LIN {X 0,Y 254.905,Z 183.243,A -85,B 0,C 180,E1 -18881.826,E2 -18881.826} C_VEL
LIN {X 0,Y 256.639,Z 184.875,A -85,B 0,C 180,E1 -18883.002,E2 -18883.002} C_VEL
LIN {X 0,Y 260.021,Z 189.343,A -85,B 0,C 180,E1 -18885.127,E2 -18885.127} C_VEL
LIN {X 0,Y 261.601,Z 191.447,A -85,B 0,C 180,E1 -18886.008,E2 -18886.008} C_VEL
LIN {X 0,Y 265.009,Z 196.05,A -85,B 0,C 180,E1 -18887.751,E2 -18887.751} C_VEL
LIN {X 0,Y 268.493,Z 201.125,A -85,B 0,C 180,E1 -18889.357,E2 -18889.357} C_VEL
LIN {X 0,Y 271.454,Z 205.94,A -85,B 0,C 180,E1 -18890.618,E2 -18890.618} C_VEL
LIN {X 0,Y 277.657,Z 217.044,A -85,B 0,C 180,E1 -18893.04,E2 -18893.04} C_VEL
LIN {X 0,Y 281.725,Z 226.048,A -85,B 0,C 180,E1 -18894.546,E2 -18894.546} C_VEL
LIN {X 0,Y 276.676,Z 285.05,A -85,B 0,C 180,E1 -18896.614,E2 -18896.614} C_VEL
LIN {X 0,Y 274.99,Z 297.648,A -85,B 0,C 180,E1 -18897.29,E2 -18897.29} C_VEL
LIN {X 0,Y 273.026,Z 309.594,A -85,B 0,C 180,E1 -18898.211,E2 -18898.211} C_VEL
LIN {X 0,Y 270.772,Z 320.185,A -85,B 0,C 180,E1 -18899.257,E2 -18899.257} C_VEL
LIN {X 0,Y 267.635,Z 332.608,A -85,B 0,C 180,E1 -18900.856,E2 -18900.856} C_VEL
LIN {X 0,Y 264.368,Z 343.674,A -85,B 0,C 180,E1 -18902.667,E2 -18902.667} C_VEL
LIN {X 0,Y 260.959,Z 353.865,A -85,B 0,C 180,E1 -18904.808,E2 -18904.808} C_VEL
LIN {X 0,Y 258.393,Z 360.832,A -85,B 0,C 180,E1 -18906.638,E2 -18906.638} C_VEL
LIN {X 0,Y 255.598,Z 368.03,A -85,B 0,C 180,E1 -18908.991,E2 -18908.991} C_VEL
LIN {X 0,Y 253.363,Z 373.364,A -85,B 0,C 180,E1 -18911.197,E2 -18911.197} C_VEL
LIN {X 0,Y 251.204,Z 378.159,A -85,B 0,C 180,E1 -18913.758,E2 -18913.758} C_VEL
LIN {X 0,Y 249.407,Z 381.995,A -85,B 0,C 180,E1 -18916.645,E2 -18916.645} C_VEL
LIN {X 0,Y 248.021,Z 384.63,A -85,B 0,C 180,E1 -18919.88,E2 -18919.88} C_VEL
LIN {X 0,Y 247.437,Z 385.342,A -85,B 0,C 180,E1 -18921.669,E2 -18921.669} C_VEL
LIN {X 0,Y 246.862,Z 385.521,A -85,B 0,C 180,E1 -18924.351,E2 -18924.351} C_VEL
LIN {X 0,Y 246.591,Z 384.531,A -85,B 0,C 180,E1 -18927.131,E2 -18927.131} C_VEL
LIN {X 0,Y 246.526,Z 383.207,A -85,B 0,C 180,E1 -18928.989,E2 -18928.989} C_VEL
LIN {X 0,Y 246.787,Z 379.889,A -85,B 0,C 180,E1 -18931.942,E2 -18931.942} C_VEL
LIN {X 0,Y 247.195,Z 375.495,A -85,B 0,C 180,E1 -18934.655,E2 -18934.655} C_VEL
LIN {X 0,Y 247.774,Z 369.505,A -85,B 0,C 180,E1 -18937.418,E2 -18937.418} C_VEL
LIN {X 0,Y 248.552,Z 362.739,A -85,B 0,C 180,E1 -18939.841,E2 -18939.841} C_VEL
LIN {X 0,Y 249.449,Z 355.299,A -85,B 0,C 180,E1 -18942.001,E2 -18942.001} C_VEL
LIN {X 0,Y 250.528,Z 346.497,A -85,B 0,C 180,E1 -18944.092,E2 -18944.092} C_VEL
LIN {X 0,Y 251.803,Z 336.515,A -85,B 0,C 180,E1 -18946.013,E2 -18946.013} C_VEL
LIN {X 0,Y 253.278,Z 324.244,A -85,B 0,C 180,E1 -18947.882,E2 -18947.882} C_VEL
LIN {X 0,Y 254.569,Z 312.848,A -85,B 0,C 180,E1 -18949.243,E2 -18949.243} C_VEL
LIN {X 0,Y 255.708,Z 299.284,A -85,B 0,C 180,E1 -18950.473,E2 -18950.473} C_VEL
LIN {X 0,Y 256.538,Z 286.069,A -85,B 0,C 180,E1 -18951.331,E2 -18951.331} C_VEL
LIN {X 0,Y 257.364,Z 267.967,A -85,B 0,C 180,E1 -18952.047,E2 -18952.047} C_VEL
LIN {X 0,Y 259.677,Z 209.083,A -85,B 0,C 180,E1 -18954.102,E2 -18954.102} C_VEL
LIN {X 0,Y 258.379,Z 202.077,A -85,B 0,C 180,E1 -18954.456,E2 -18954.456} C_VEL
LIN {X 0,Y 249.422,Z 174.029,A -85,B 0,C 180,E1 -18956.245,E2 -18956.245} C_VEL
LIN {X 0,Y 249.088,Z 172.457,A -85,B 0,C 180,E1 -18956.92,E2 -18956.92} C_VEL
LIN {X 0,Y 249.039,Z 172.462,A -85,B 0,C 180,E1 -18961.33,E2 -18961.33} C_VEL
LIN {X 0,Y 249.06,Z 172.46,A -85,B 0,C 180,E1 -18964.957,E2 -18964.957} C_VEL
LIN {X 0,Y 249.055,Z 172.461,A -85,B 0,C 180,E1 -18968.627,E2 -18968.627} C_VEL
LIN {X 0,Y 249.162,Z 172.448,A -85,B 0,C 180,E1 -18973.615,E2 -18973.615} C_VEL
LIN {X 0,Y 249.223,Z 172.44,A -85,B 0,C 180,E1 -18978.614,E2 -18978.614} C_VEL
LIN {X 0,Y 249.435,Z 172.416,A -85,B 0,C 180,E1 -18981.9,E2 -18981.9} C_VEL
LIN {X 0,Y 249.264,Z 172.434,A -85,B 0,C 180,E1 -18985.146,E2 -18985.146} C_VEL
LIN {X 0,Y 249.661,Z 172.384,A -85,B 0,C 180,E1 -18988.386,E2 -18988.386} C_VEL
LIN {X 0,Y 249.66,Z 172.385,A -85,B 0,C 180,E1 -18991.612,E2 -18991.612} C_VEL
LIN {X 0,Y 249.428,Z 172.412,A -85,B 0,C 180,E1 -18996.47,E2 -18996.47} C_VEL
LIN {X 0,Y 249.335,Z 172.427,A -85,B 0,C 180,E1 -18999.735,E2 -18999.735} C_VEL
LIN {X 0,Y 249.147,Z 172.448,A -85,B 0,C 180,E1 -19004.705,E2 -19004.705} C_VEL
LIN {X 0,Y 249.079,Z 172.456,A -85,B 0,C 180,E1 -19008.08,E2 -19008.08} C_VEL
LIN {X 0,Y 249.043,Z 172.464,A -85,B 0,C 180,E1 -19011.521,E2 -19011.521} C_VEL
LIN {X 0,Y 249.047,Z 172.462,A -85,B 0,C 180,E1 -19015.44,E2 -19015.44} C_VEL
LIN {X 0,Y 249.036,Z 172.464,A -85,B 0,C 180,E1 -19018.972,E2 -19018.972} C_VEL
LIN {X 0,Y 249.026,Z 172.462,A -85,B 0,C 180,E1 -19022.425,E2 -19022.425} C_VEL
LIN {X 0,Y 249.025,Z 172.463,A -85,B 0,C 180,E1 -19026.344,E2 -19026.344} C_VEL
LIN {X 0,Y 248.976,Z 172.47,A -85,B 0,C 180,E1 -19030.482,E2 -19030.482} C_VEL
LIN {X 0,Y 248.959,Z 172.475,A -85,B 0,C 180,E1 -19034.887,E2 -19034.887} C_VEL
LIN {X 0,Y 248.976,Z 172.47,A -85,B 0,C 180,E1 -19037.353,E2 -19037.353} C_VEL
LIN {X 0,Y 249.036,Z 172.462,A -85,B 0,C 180,E1 -19042.2,E2 -19042.2} C_VEL
LIN {X 0,Y 249.039,Z 172.461,A -85,B 0,C 180,E1 -19045.638,E2 -19045.638} C_VEL
LIN {X 0,Y 248.997,Z 172.465,A -85,B 0,C 180,E1 -19049.465,E2 -19049.465} C_VEL
LIN {X 0,Y 249.016,Z 172.465,A -85,B 0,C 180,E1 -19053.155,E2 -19053.155} C_VEL
LIN {X 0,Y 249,Z 172.466,A -85,B 0,C 180,E1 -19056.724,E2 -19056.724} C_VEL
LIN {X 0,Y 249.037,Z 172.464,A -85,B 0,C 180,E1 -19060.205,E2 -19060.205} C_VEL
LIN {X 0,Y 249.152,Z 172.447,A -85,B 0,C 180,E1 -19063.615,E2 -19063.615} C_VEL
LIN {X 0,Y 249.211,Z 172.441,A -85,B 0,C 180,E1 -19068.614,E2 -19068.614} C_VEL
LIN {X 0,Y 249.425,Z 172.416,A -85,B 0,C 180,E1 -19071.901,E2 -19071.901} C_VEL
LIN {X 0,Y 249.254,Z 172.433,A -85,B 0,C 180,E1 -19075.147,E2 -19075.147} C_VEL
LIN {X 0,Y 249.65,Z 172.387,A -85,B 0,C 180,E1 -19078.386,E2 -19078.386} C_VEL
LIN {X 0,Y 249.649,Z 172.386,A -85,B 0,C 180,E1 -19081.613,E2 -19081.613} C_VEL
LIN {X 0,Y 249.418,Z 172.415,A -85,B 0,C 180,E1 -19086.471,E2 -19086.471} C_VEL
LIN {X 0,Y 249.325,Z 172.428,A -85,B 0,C 180,E1 -19089.737,E2 -19089.737} C_VEL
LIN {X 0,Y 249.138,Z 172.449,A -85,B 0,C 180,E1 -19094.707,E2 -19094.707} C_VEL
LIN {X 0,Y 249.119,Z 172.448,A -85,B 0,C 180,E1 -19095.622,E2 -19095.622} C_VEL
LIN {X 0,Y 248.461,Z 172.535,A -85,B 0,C 180,E1 -19096.971,E2 -19096.971} C_VEL
LIN {X 0,Y 245.577,Z 172.894,A -85,B 0,C 180,E1 -19099.169,E2 -19099.169} C_VEL
LIN {X 0,Y 243.104,Z 173.201,A -85,B 0,C 180,E1 -19100.959,E2 -19100.959} C_VEL
LIN {X 0,Y 242.028,Z 173.335,A -85,B 0,C 180,E1 -19102.349,E2 -19102.349} C_VEL
LIN {X 0,Y 241.933,Z 173.344,A -85,B 0,C 180,E1 -19102.821,E2 -19102.821} C_VEL
LIN {X 0,Y 241.98,Z 173.341,A -85,B 0,C 180,E1 -19105.827,E2 -19105.827} C_VEL
LIN {X 0,Y 241.962,Z 173.345,A -85,B 0,C 180,E1 -19109.589,E2 -19109.589} C_VEL
LIN {X 0,Y 241.973,Z 173.343,A -85,B 0,C 180,E1 -19113.494,E2 -19113.494} C_VEL
LIN {X 0,Y 241.977,Z 173.342,A -85,B 0,C 180,E1 -19117.584,E2 -19117.584} C_VEL
LIN {X 0,Y 241.902,Z 173.35,A -85,B 0,C 180,E1 -19121.93,E2 -19121.93} C_VEL
LIN {X 0,Y 241.895,Z 173.354,A -85,B 0,C 180,E1 -19126.581,E2 -19126.581} C_VEL
LIN {X 0,Y 241.988,Z 173.34,A -85,B 0,C 180,E1 -19131.642,E2 -19131.642} C_VEL
LIN {X 0,Y 242.069,Z 173.515,A -85,B 0,C 180,E1 -19136.148,E2 -19136.148} C_VEL
LIN {X 0,Y 244.15,Z 184.245,A -85,B 0,C 180,E1 -19140.267,E2 -19140.267} C_VEL
LIN {X 0,Y 244.801,Z 187.444,A -85,B 0,C 180,E1 -19141.446,E2 -19141.446} C_VEL
LIN {X 0,Y 248.272,Z 199.557,A -85,B 0,C 180,E1 -19142.193,E2 -19142.193} C_VEL
LIN {X 0,Y 252.252,Z 234.822,A -85,B 0,C 180,E1 -19143.86,E2 -19143.86} C_VEL
LIN {X 0,Y 249.825,Z 295.765,A -85,B 0,C 180,E1 -19146.093,E2 -19146.093} C_VEL
LIN {X 0,Y 248.844,Z 309.841,A -85,B 0,C 180,E1 -19146.931,E2 -19146.931} C_VEL
LIN {X 0,Y 247.722,Z 321.604,A -85,B 0,C 180,E1 -19147.921,E2 -19147.921} C_VEL
LIN {X 0,Y 246.377,Z 334.101,A -85,B 0,C 180,E1 -19149.331,E2 -19149.331} C_VEL
LIN {X 0,Y 244.925,Z 345.362,A -85,B 0,C 180,E1 -19150.951,E2 -19150.951} C_VEL
LIN {X 0,Y 243.54,Z 355.921,A -85,B 0,C 180,E1 -19152.864,E2 -19152.864} C_VEL
LIN {X 0,Y 242.419,Z 364.893,A -85,B 0,C 180,E1 -19154.877,E2 -19154.877} C_VEL
LIN {X 0,Y 241.251,Z 373.932,A -85,B 0,C 180,E1 -19157.381,E2 -19157.381} C_VEL
LIN {X 0,Y 240.534,Z 381.125,A -85,B 0,C 180,E1 -19159.905,E2 -19159.905} C_VEL
LIN {X 0,Y 240.116,Z 386.836,A -85,B 0,C 180,E1 -19162.433,E2 -19162.433} C_VEL
LIN {X 0,Y 239.919,Z 391.263,A -85,B 0,C 180,E1 -19164.96,E2 -19164.96} C_VEL
LIN {X 0,Y 239.892,Z 393.581,A -85,B 0,C 180,E1 -19166.642,E2 -19166.642} C_VEL
LIN {X 0,Y 239.92,Z 395.406,A -85,B 0,C 180,E1 -19168.323,E2 -19168.323} C_VEL
LIN {X 0,Y 239.916,Z 396.747,A -85,B 0,C 180,E1 -19170.001,E2 -19170.001} C_VEL
LIN {X 0,Y 239.893,Z 397.668,A -85,B 0,C 180,E1 -19171.68,E2 -19171.68} C_VEL
LIN {X 0,Y 239.775,Z 398.264,A -85,B 0,C 180,E1 -19174.748,E2 -19174.748} C_VEL
LIN {X 0,Y 239.96,Z 397.891,A -85,B 0,C 180,E1 -19176.729,E2 -19176.729} C_VEL
LIN {X 0,Y 240.757,Z 396.027,A -85,B 0,C 180,E1 -19180.089,E2 -19180.089} C_VEL
LIN {X 0,Y 241.785,Z 393.519,A -85,B 0,C 180,E1 -19182.593,E2 -19182.593} C_VEL
LIN {X 0,Y 243.188,Z 390.027,A -85,B 0,C 180,E1 -19185.077,E2 -19185.077} C_VEL
LIN {X 0,Y 245.352,Z 385.49,A -85,B 0,C 180,E1 -19187.505,E2 -19187.505} C_VEL
LIN {X 0,Y 248.14,Z 378.736,A -85,B 0,C 180,E1 -19190.302,E2 -19190.302} C_VEL
LIN {X 0,Y 250.933,Z 371.563,A -85,B 0,C 180,E1 -19192.608,E2 -19192.608} C_VEL
LIN {X 0,Y 254.355,Z 362.426,A -85,B 0,C 180,E1 -19194.922,E2 -19194.922} C_VEL
LIN {X 0,Y 257.945,Z 352.315,A -85,B 0,C 180,E1 -19196.936,E2 -19196.936} C_VEL
LIN {X 0,Y 261.529,Z 340.93,A -85,B 0,C 180,E1 -19198.71,E2 -19198.71} C_VEL
LIN {X 0,Y 264.574,Z 329.639,A -85,B 0,C 180,E1 -19200.093,E2 -19200.093} C_VEL
LIN {X 0,Y 267.49,Z 316.966,A -85,B 0,C 180,E1 -19201.26,E2 -19201.26} C_VEL
LIN {X 0,Y 270.042,Z 303.682,A -85,B 0,C 180,E1 -19202.135,E2 -19202.135} C_VEL
LIN {X 0,Y 271.757,Z 289.867,A -85,B 0,C 180,E1 -19202.785,E2 -19202.785} C_VEL
LIN {X 0,Y 275.895,Z 241.621,A -85,B 0,C 180,E1 -19204.522,E2 -19204.522} C_VEL
LIN {X 0,Y 275,Z 233.168,A -85,B 0,C 180,E1 -19205.232,E2 -19205.232} C_VEL
LIN {X 0,Y 271.422,Z 224.233,A -85,B 0,C 180,E1 -19206.741,E2 -19206.741} C_VEL
LIN {X 0,Y 266.748,Z 214.805,A -85,B 0,C 180,E1 -19208.789,E2 -19208.789} C_VEL
LIN {X 0,Y 264.621,Z 210.789,A -85,B 0,C 180,E1 -19209.822,E2 -19209.822} C_VEL
LIN {X 0,Y 262.005,Z 206.304,A -85,B 0,C 180,E1 -19211.117,E2 -19211.117} C_VEL
LIN {X 0,Y 258.799,Z 200.968,A -85,B 0,C 180,E1 -19212.915,E2 -19212.915} C_VEL
LIN {X 0,Y 254.883,Z 194.985,A -85,B 0,C 180,E1 -19215.414,E2 -19215.414} C_VEL
LIN {X 0,Y 250.245,Z 188.473,A -85,B 0,C 180,E1 -19219.227,E2 -19219.227} C_VEL
LIN {X 0,Y 246.767,Z 184.055,A -85,B 0,C 180,E1 -19223.65,E2 -19223.65} C_VEL
LIN {X 0,Y 245.502,Z 182.109,A -85,B 0,C 180,E1 -19227.05,E2 -19227.05} C_VEL
LIN {X 0,Y 245.288,Z 181.573,A -85,B 0,C 180,E1 -19229.269,E2 -19229.269} C_VEL
LIN {X 0,Y 245.694,Z 181.933,A -85,B 0,C 180,E1 -19232.047,E2 -19232.047} C_VEL
LIN {X 0,Y 247.908,Z 184.21,A -85,B 0,C 180,E1 -19236.395,E2 -19236.395} C_VEL
LIN {X 0,Y 250.046,Z 185.965,A -85,B 0,C 180,E1 -19238.785,E2 -19238.785} C_VEL
LIN {X 0,Y 253.178,Z 190.055,A -85,B 0,C 180,E1 -19241.593,E2 -19241.593} C_VEL
LIN {X 0,Y 254.488,Z 191.344,A -85,B 0,C 180,E1 -19242.517,E2 -19242.517} C_VEL
LIN {X 0,Y 258.027,Z 196.028,A -85,B 0,C 180,E1 -19244.837,E2 -19244.837} C_VEL
LIN {X 0,Y 262.472,Z 202.382,A -85,B 0,C 180,E1 -19247.297,E2 -19247.297} C_VEL
LIN {X 0,Y 265.653,Z 207.183,A -85,B 0,C 180,E1 -19248.822,E2 -19248.822} C_VEL
LIN {X 0,Y 268.38,Z 211.88,A -85,B 0,C 180,E1 -19250.079,E2 -19250.079} C_VEL
LIN {X 0,Y 274.089,Z 222.548,A -85,B 0,C 180,E1 -19252.449,E2 -19252.449} C_VEL
LIN {X 0,Y 276.862,Z 228.786,A -85,B 0,C 180,E1 -19253.522,E2 -19253.522} C_VEL
LIN {X 0,Y 271.748,Z 285.239,A -85,B 0,C 180,E1 -19255.55,E2 -19255.55} C_VEL
LIN {X 0,Y 269.887,Z 298.289,A -85,B 0,C 180,E1 -19256.268,E2 -19256.268} C_VEL
LIN {X 0,Y 267.768,Z 310.372,A -85,B 0,C 180,E1 -19257.216,E2 -19257.216} C_VEL
LIN {X 0,Y 265.372,Z 320.961,A -85,B 0,C 180,E1 -19258.284,E2 -19258.284} C_VEL
LIN {X 0,Y 262.265,Z 332.663,A -85,B 0,C 180,E1 -19259.808,E2 -19259.808} C_VEL
LIN {X 0,Y 258.966,Z 343.263,A -85,B 0,C 180,E1 -19261.555,E2 -19261.555} C_VEL
LIN {X 0,Y 255.612,Z 352.681,A -85,B 0,C 180,E1 -19263.53,E2 -19263.53} C_VEL
LIN {X 0,Y 251.986,Z 362.014,A -85,B 0,C 180,E1 -19266.004,E2 -19266.004} C_VEL
LIN {X 0,Y 248.799,Z 369.538,A -85,B 0,C 180,E1 -19268.625,E2 -19268.625} C_VEL
LIN {X 0,Y 245.854,Z 375.898,A -85,B 0,C 180,E1 -19271.543,E2 -19271.543} C_VEL
LIN {X 0,Y 243.79,Z 380.082,A -85,B 0,C 180,E1 -19274.185,E2 -19274.185} C_VEL
LIN {X 0,Y 242.176,Z 383.099,A -85,B 0,C 180,E1 -19276.871,E2 -19276.871} C_VEL
LIN {X 0,Y 241.372,Z 384.47,A -85,B 0,C 180,E1 -19278.681,E2 -19278.681} C_VEL
LIN {X 0,Y 240.58,Z 385.479,A -85,B 0,C 180,E1 -19280.799,E2 -19280.799} C_VEL
LIN {X 0,Y 240.168,Z 385.781,A -85,B 0,C 180,E1 -19282.36,E2 -19282.36} C_VEL
LIN {X 0,Y 239.708,Z 385.624,A -85,B 0,C 180,E1 -19284.645,E2 -19284.645} C_VEL
LIN {X 0,Y 239.532,Z 385.104,A -85,B 0,C 180,E1 -19286.111,E2 -19286.111} C_VEL
LIN {X 0,Y 239.438,Z 383.75,A -85,B 0,C 180,E1 -19288.287,E2 -19288.287} C_VEL
LIN {X 0,Y 239.541,Z 381.245,A -85,B 0,C 180,E1 -19290.839,E2 -19290.839} C_VEL
LIN {X 0,Y 239.971,Z 376.997,A -85,B 0,C 180,E1 -19293.811,E2 -19293.811} C_VEL
LIN {X 0,Y 240.509,Z 371.044,A -85,B 0,C 180,E1 -19296.802,E2 -19296.802} C_VEL
LIN {X 0,Y 241.244,Z 364.525,A -85,B 0,C 180,E1 -19299.339,E2 -19299.339} C_VEL
LIN {X 0,Y 242.257,Z 356.378,A -85,B 0,C 180,E1 -19301.855,E2 -19301.855} C_VEL
LIN {X 0,Y 243.418,Z 347.106,A -85,B 0,C 180,E1 -19304.151,E2 -19304.151} C_VEL
LIN {X 0,Y 244.749,Z 336.839,A -85,B 0,C 180,E1 -19306.201,E2 -19306.201} C_VEL
LIN {X 0,Y 246.095,Z 325.865,A -85,B 0,C 180,E1 -19307.947,E2 -19307.947} C_VEL
LIN {X 0,Y 247.486,Z 313.985,A -85,B 0,C 180,E1 -19309.447,E2 -19309.447} C_VEL
LIN {X 0,Y 248.646,Z 301.024,A -85,B 0,C 180,E1 -19310.693,E2 -19310.693} C_VEL
LIN {X 0,Y 249.585,Z 287.032,A -85,B 0,C 180,E1 -19311.663,E2 -19311.663} C_VEL
LIN {X 0,Y 250.44,Z 270.442,A -85,B 0,C 180,E1 -19312.364,E2 -19312.364} C_VEL
LIN {X 0,Y 252.892,Z 210.015,A -85,B 0,C 180,E1 -19314.539,E2 -19314.539} C_VEL
LIN {X 0,Y 251.787,Z 204.045,A -85,B 0,C 180,E1 -19314.85,E2 -19314.85} C_VEL
LIN {X 0,Y 242.629,Z 175.689,A -85,B 0,C 180,E1 -19316.676,E2 -19316.676} C_VEL
LIN {X 0,Y 242.213,Z 174.177,A -85,B 0,C 180,E1 -19316.819,E2 -19316.819} C_VEL
LIN {X 0,Y 242.034,Z 173.334,A -85,B 0,C 180,E1 -19317.294,E2 -19317.294} C_VEL
LIN {X 0,Y 241.976,Z 173.345,A -85,B 0,C 180,E1 -19320.615,E2 -19320.615} C_VEL
LIN {X 0,Y 242.001,Z 173.342,A -85,B 0,C 180,E1 -19324.196,E2 -19324.196} C_VEL
LIN {X 0,Y 241.99,Z 173.343,A -85,B 0,C 180,E1 -19328.337,E2 -19328.337} C_VEL
LIN {X 0,Y 242.11,Z 173.325,A -85,B 0,C 180,E1 -19333.323,E2 -19333.323} C_VEL
LIN {X 0,Y 242.157,Z 173.322,A -85,B 0,C 180,E1 -19338.277,E2 -19338.277} C_VEL
LIN {X 0,Y 242.385,Z 173.292,A -85,B 0,C 180,E1 -19341.663,E2 -19341.663} C_VEL
LIN {X 0,Y 242.404,Z 173.289,A -85,B 0,C 180,E1 -19343.339,E2 -19343.339} C_VEL
LIN {X 0,Y 242.621,Z 173.261,A -85,B 0,C 180,E1 -19348.339,E2 -19348.339} C_VEL
LIN {X 0,Y 242.62,Z 173.263,A -85,B 0,C 180,E1 -19351.658,E2 -19351.658} C_VEL
LIN {X 0,Y 242.398,Z 173.288,A -85,B 0,C 180,E1 -19356.658,E2 -19356.658} C_VEL
LIN {X 0,Y 242.262,Z 173.306,A -85,B 0,C 180,E1 -19360.022,E2 -19360.022} C_VEL
LIN {X 0,Y 242.106,Z 173.326,A -85,B 0,C 180,E1 -19365.143,E2 -19365.143} C_VEL
LIN {X 0,Y 242.017,Z 173.335,A -85,B 0,C 180,E1 -19368.627,E2 -19368.627} C_VEL
LIN {X 0,Y 241.973,Z 173.341,A -85,B 0,C 180,E1 -19372.182,E2 -19372.182} C_VEL
LIN {X 0,Y 241.987,Z 173.339,A -85,B 0,C 180,E1 -19375.825,E2 -19375.825} C_VEL
LIN {X 0,Y 241.968,Z 173.344,A -85,B 0,C 180,E1 -19379.587,E2 -19379.587} C_VEL
LIN {X 0,Y 241.978,Z 173.341,A -85,B 0,C 180,E1 -19383.491,E2 -19383.491} C_VEL
LIN {X 0,Y 241.981,Z 173.342,A -85,B 0,C 180,E1 -19387.581,E2 -19387.581} C_VEL
LIN {X 0,Y 241.905,Z 173.347,A -85,B 0,C 180,E1 -19391.927,E2 -19391.927} C_VEL
LIN {X 0,Y 241.897,Z 173.354,A -85,B 0,C 180,E1 -19396.578,E2 -19396.578} C_VEL
LIN {X 0,Y 241.988,Z 173.339,A -85,B 0,C 180,E1 -19401.64,E2 -19401.64} C_VEL
LIN {X 0,Y 241.975,Z 173.344,A -85,B 0,C 180,E1 -19404.486,E2 -19404.486} C_VEL
LIN {X 0,Y 241.948,Z 173.346,A -85,B 0,C 180,E1 -19408.475,E2 -19408.475} C_VEL
LIN {X 0,Y 241.955,Z 173.346,A -85,B 0,C 180,E1 -19412.306,E2 -19412.306} C_VEL
LIN {X 0,Y 241.976,Z 173.342,A -85,B 0,C 180,E1 -19416.007,E2 -19416.007} C_VEL
LIN {X 0,Y 241.977,Z 173.341,A -85,B 0,C 180,E1 -19419.602,E2 -19419.602} C_VEL
LIN {X 0,Y 242.1,Z 173.325,A -85,B 0,C 180,E1 -19423.323,E2 -19423.323} C_VEL
LIN {X 0,Y 242.145,Z 173.324,A -85,B 0,C 180,E1 -19428.277,E2 -19428.277} C_VEL
LIN {X 0,Y 242.374,Z 173.293,A -85,B 0,C 180,E1 -19431.663,E2 -19431.663} C_VEL
LIN {X 0,Y 242.393,Z 173.288,A -85,B 0,C 180,E1 -19433.34,E2 -19433.34} C_VEL
LIN {X 0,Y 242.61,Z 173.264,A -85,B 0,C 180,E1 -19438.34,E2 -19438.34} C_VEL
LIN {X 0,Y 242.609,Z 173.264,A -85,B 0,C 180,E1 -19441.66,E2 -19441.66} C_VEL
LIN {X 0,Y 242.389,Z 173.29,A -85,B 0,C 180,E1 -19446.66,E2 -19446.66} C_VEL
LIN {X 0,Y 242.253,Z 173.306,A -85,B 0,C 180,E1 -19450.024,E2 -19450.024} C_VEL
LIN {X 0,Y 242.097,Z 173.327,A -85,B 0,C 180,E1 -19455.145,E2 -19455.145} C_VEL
LIN {X 0,Y 242.009,Z 173.335,A -85,B 0,C 180,E1 -19458.629,E2 -19458.629} C_VEL
LIN {X 0,Y 241.933,Z 173.344,A -85,B 0,C 180,E1 -19462.821,E2 -19462.821} C_VEL
LIN {X 0,Y 241.254,Z 173.432,A -85,B 0,C 180,E1 -19464.209,E2 -19464.209} C_VEL
LIN {X 0,Y 238.431,Z 173.781,A -85,B 0,C 180,E1 -19466.475,E2 -19466.475} C_VEL
LIN {X 0,Y 236.033,Z 174.082,A -85,B 0,C 180,E1 -19468.321,E2 -19468.321} C_VEL
LIN {X 0,Y 234.991,Z 174.213,A -85,B 0,C 180,E1 -19469.752,E2 -19469.752} C_VEL
LIN {X 0,Y 234.898,Z 174.223,A -85,B 0,C 180,E1 -19470.237,E2 -19470.237} C_VEL
LIN {X 0,Y 234.935,Z 174.222,A -85,B 0,C 180,E1 -19473.114,E2 -19473.114} C_VEL
LIN {X 0,Y 234.909,Z 174.219,A -85,B 0,C 180,E1 -19476.752,E2 -19476.752} C_VEL
LIN {X 0,Y 234.906,Z 174.224,A -85,B 0,C 180,E1 -19478.936,E2 -19478.936} C_VEL
LIN {X 0,Y 234.848,Z 174.231,A -85,B 0,C 180,E1 -19483.495,E2 -19483.495} C_VEL
LIN {X 0,Y 234.848,Z 174.231,A -85,B 0,C 180,E1 -19486.507,E2 -19486.507} C_VEL
LIN {X 0,Y 234.913,Z 174.224,A -85,B 0,C 180,E1 -19491.08,E2 -19491.08} C_VEL
LIN {X 0,Y 234.974,Z 174.215,A -85,B 0,C 180,E1 -19495.742,E2 -19495.742} C_VEL
LIN {X 0,Y 236.966,Z 184.264,A -85,B 0,C 180,E1 -19499.724,E2 -19499.724} C_VEL
LIN {X 0,Y 237.523,Z 187.283,A -85,B 0,C 180,E1 -19500.863,E2 -19500.863} C_VEL
LIN {X 0,Y 241.639,Z 201.481,A -85,B 0,C 180,E1 -19501.776,E2 -19501.776} C_VEL
LIN {X 0,Y 245.429,Z 235.077,A -85,B 0,C 180,E1 -19503.419,E2 -19503.419} C_VEL
LIN {X 0,Y 242.873,Z 296.425,A -85,B 0,C 180,E1 -19505.763,E2 -19505.763} C_VEL
LIN {X 0,Y 241.803,Z 310.913,A -85,B 0,C 180,E1 -19506.673,E2 -19506.673} C_VEL
LIN {X 0,Y 240.408,Z 324.215,A -85,B 0,C 180,E1 -19507.892,E2 -19507.892} C_VEL
LIN {X 0,Y 239.075,Z 336.161,A -85,B 0,C 180,E1 -19509.345,E2 -19509.345} C_VEL
LIN {X 0,Y 237.67,Z 346.965,A -85,B 0,C 180,E1 -19511.019,E2 -19511.019} C_VEL
LIN {X 0,Y 236.276,Z 357.877,A -85,B 0,C 180,E1 -19513.143,E2 -19513.143} C_VEL
LIN {X 0,Y 235.101,Z 366.753,A -85,B 0,C 180,E1 -19515.282,E2 -19515.282} C_VEL
LIN {X 0,Y 233.99,Z 375.327,A -85,B 0,C 180,E1 -19517.865,E2 -19517.865} C_VEL
LIN {X 0,Y 233.339,Z 382.22,A -85,B 0,C 180,E1 -19520.466,E2 -19520.466} C_VEL
LIN {X 0,Y 232.974,Z 387.672,A -85,B 0,C 180,E1 -19523.071,E2 -19523.071} C_VEL
LIN {X 0,Y 232.779,Z 392.073,A -85,B 0,C 180,E1 -19525.832,E2 -19525.832} C_VEL
LIN {X 0,Y 232.853,Z 394.895,A -85,B 0,C 180,E1 -19528.272,E2 -19528.272} C_VEL
LIN {X 0,Y 232.849,Z 396.323,A -85,B 0,C 180,E1 -19530.001,E2 -19530.001} C_VEL
LIN {X 0,Y 232.822,Z 397.301,A -85,B 0,C 180,E1 -19531.731,E2 -19531.731} C_VEL
LIN {X 0,Y 232.731,Z 398.041,A -85,B 0,C 180,E1 -19535.199,E2 -19535.199} C_VEL
LIN {X 0,Y 232.898,Z 397.786,A -85,B 0,C 180,E1 -19536.934,E2 -19536.934} C_VEL
LIN {X 0,Y 233.754,Z 396.054,A -85,B 0,C 180,E1 -19540.394,E2 -19540.394} C_VEL
LIN {X 0,Y 234.424,Z 394.601,A -85,B 0,C 180,E1 -19542.116,E2 -19542.116} C_VEL
LIN {X 0,Y 235.807,Z 391.606,A -85,B 0,C 180,E1 -19544.676,E2 -19544.676} C_VEL
LIN {X 0,Y 237.807,Z 387.594,A -85,B 0,C 180,E1 -19547.191,E2 -19547.191} C_VEL
LIN {X 0,Y 240.226,Z 382.472,A -85,B 0,C 180,E1 -19549.662,E2 -19549.662} C_VEL
LIN {X 0,Y 243.347,Z 375.051,A -85,B 0,C 180,E1 -19552.455,E2 -19552.455} C_VEL
LIN {X 0,Y 246.815,Z 366.854,A -85,B 0,C 180,E1 -19554.836,E2 -19554.836} C_VEL
LIN {X 0,Y 250.079,Z 358.685,A -85,B 0,C 180,E1 -19556.723,E2 -19556.723} C_VEL
LIN {X 0,Y 253.618,Z 348.854,A -85,B 0,C 180,E1 -19558.557,E2 -19558.557} C_VEL
LIN {X 0,Y 257.078,Z 337.949,A -85,B 0,C 180,E1 -19560.156,E2 -19560.156} C_VEL
LIN {X 0,Y 260.279,Z 326.083,A -85,B 0,C 180,E1 -19561.546,E2 -19561.546} C_VEL
LIN {X 0,Y 263.256,Z 313.617,A -85,B 0,C 180,E1 -19562.613,E2 -19562.613} C_VEL
LIN {X 0,Y 265.824,Z 299.296,A -85,B 0,C 180,E1 -19563.499,E2 -19563.499} C_VEL
LIN {X 0,Y 267.505,Z 284.583,A -85,B 0,C 180,E1 -19564.11,E2 -19564.11} C_VEL
LIN {X 0,Y 271.233,Z 242.722,A -85,B 0,C 180,E1 -19565.634,E2 -19565.634} C_VEL
LIN {X 0,Y 270.589,Z 236.589,A -85,B 0,C 180,E1 -19566.192,E2 -19566.192} C_VEL
LIN {X 0,Y 267.522,Z 228.685,A -85,B 0,C 180,E1 -19567.596,E2 -19567.596} C_VEL
LIN {X 0,Y 263.147,Z 219.479,A -85,B 0,C 180,E1 -19569.681,E2 -19569.681} C_VEL
LIN {X 0,Y 259.324,Z 212.341,A -85,B 0,C 180,E1 -19571.689,E2 -19571.689} C_VEL
LIN {X 0,Y 256.114,Z 206.872,A -85,B 0,C 180,E1 -19573.584,E2 -19573.584} C_VEL
LIN {X 0,Y 252.574,Z 201.25,A -85,B 0,C 180,E1 -19576.012,E2 -19576.012} C_VEL
LIN {X 0,Y 248.508,Z 195.193,A -85,B 0,C 180,E1 -19579.571,E2 -19579.571} C_VEL
LIN {X 0,Y 245.41,Z 191.101,A -85,B 0,C 180,E1 -19583.672,E2 -19583.672} C_VEL
LIN {X 0,Y 244.227,Z 189.186,A -85,B 0,C 180,E1 -19586.856,E2 -19586.856} C_VEL
LIN {X 0,Y 244.008,Z 188.574,A -85,B 0,C 180,E1 -19589.779,E2 -19589.779} C_VEL
LIN {X 0,Y 244.66,Z 189.279,A -85,B 0,C 180,E1 -19592.938,E2 -19592.938} C_VEL
LIN {X 0,Y 247.691,Z 192.068,A -85,B 0,C 180,E1 -19597.72,E2 -19597.72} C_VEL
LIN {X 0,Y 248.518,Z 193.051,A -85,B 0,C 180,E1 -19598.657,E2 -19598.657} C_VEL
LIN {X 0,Y 251.307,Z 196.727,A -85,B 0,C 180,E1 -19601.239,E2 -19601.239} C_VEL
LIN {X 0,Y 252.564,Z 198.101,A -85,B 0,C 180,E1 -19602.176,E2 -19602.176} C_VEL
LIN {X 0,Y 256.458,Z 203.511,A -85,B 0,C 180,E1 -19604.811,E2 -19604.811} C_VEL
LIN {X 0,Y 260.014,Z 208.745,A -85,B 0,C 180,E1 -19606.842,E2 -19606.842} C_VEL
LIN {X 0,Y 263.379,Z 214.14,A -85,B 0,C 180,E1 -19608.544,E2 -19608.544} C_VEL
LIN {X 0,Y 268.016,Z 222.774,A -85,B 0,C 180,E1 -19610.704,E2 -19610.704} C_VEL
LIN {X 0,Y 270.838,Z 228.645,A -85,B 0,C 180,E1 -19611.917,E2 -19611.917} C_VEL
LIN {X 0,Y 272.055,Z 231.415,A -85,B 0,C 180,E1 -19612.439,E2 -19612.439} C_VEL
LIN {X 0,Y 266.878,Z 286.468,A -85,B 0,C 180,E1 -19614.475,E2 -19614.475} C_VEL
LIN {X 0,Y 264.826,Z 299.951,A -85,B 0,C 180,E1 -19615.243,E2 -19615.243} C_VEL
LIN {X 0,Y 262.667,Z 311.193,A -85,B 0,C 180,E1 -19616.165,E2 -19616.165} C_VEL
LIN {X 0,Y 259.879,Z 322.629,A -85,B 0,C 180,E1 -19617.37,E2 -19617.37} C_VEL
LIN {X 0,Y 256.401,Z 334.728,A -85,B 0,C 180,E1 -19619.019,E2 -19619.019} C_VEL
LIN {X 0,Y 253.034,Z 344.688,A -85,B 0,C 180,E1 -19620.741,E2 -19620.741} C_VEL
LIN {X 0,Y 249.429,Z 354.232,A -85,B 0,C 180,E1 -19622.827,E2 -19622.827} C_VEL
LIN {X 0,Y 246.175,Z 361.873,A -85,B 0,C 180,E1 -19624.914,E2 -19624.914} C_VEL
LIN {X 0,Y 242.906,Z 369.176,A -85,B 0,C 180,E1 -19627.482,E2 -19627.482} C_VEL
LIN {X 0,Y 240.042,Z 375.012,A -85,B 0,C 180,E1 -19630.118,E2 -19630.118} C_VEL
LIN {X 0,Y 237.731,Z 379.318,A -85,B 0,C 180,E1 -19632.685,E2 -19632.685} C_VEL
LIN {X 0,Y 235.767,Z 382.763,A -85,B 0,C 180,E1 -19635.563,E2 -19635.563} C_VEL
LIN {X 0,Y 234.801,Z 384.305,A -85,B 0,C 180,E1 -19637.417,E2 -19637.417} C_VEL
LIN {X 0,Y 234,Z 385.341,A -85,B 0,C 180,E1 -19639.292,E2 -19639.292} C_VEL
LIN {X 0,Y 233.369,Z 385.933,A -85,B 0,C 180,E1 -19641.186,E2 -19641.186} C_VEL
LIN {X 0,Y 232.883,Z 386.004,A -85,B 0,C 180,E1 -19643.099,E2 -19643.099} C_VEL
LIN {X 0,Y 232.543,Z 385.571,A -85,B 0,C 180,E1 -19645.032,E2 -19645.032} C_VEL
LIN {X 0,Y 232.366,Z 384.64,A -85,B 0,C 180,E1 -19646.981,E2 -19646.981} C_VEL
LIN {X 0,Y 232.362,Z 382.163,A -85,B 0,C 180,E1 -19649.938,E2 -19649.938} C_VEL
LIN {X 0,Y 232.764,Z 378.348,A -85,B 0,C 180,E1 -19652.922,E2 -19652.922} C_VEL
LIN {X 0,Y 233.142,Z 373.821,A -85,B 0,C 180,E1 -19655.518,E2 -19655.518} C_VEL
LIN {X 0,Y 233.777,Z 367.735,A -85,B 0,C 180,E1 -19658.228,E2 -19658.228} C_VEL
LIN {X 0,Y 234.612,Z 360.876,A -85,B 0,C 180,E1 -19660.659,E2 -19660.659} C_VEL
LIN {X 0,Y 235.57,Z 353.344,A -85,B 0,C 180,E1 -19662.833,E2 -19662.833} C_VEL
LIN {X 0,Y 236.834,Z 343.572,A -85,B 0,C 180,E1 -19665.126,E2 -19665.126} C_VEL
LIN {X 0,Y 238.258,Z 332.668,A -85,B 0,C 180,E1 -19667.183,E2 -19667.183} C_VEL
LIN {X 0,Y 239.801,Z 320.358,A -85,B 0,C 180,E1 -19668.998,E2 -19668.998} C_VEL
LIN {X 0,Y 241.073,Z 308.657,A -85,B 0,C 180,E1 -19670.349,E2 -19670.349} C_VEL
LIN {X 0,Y 242.14,Z 295.755,A -85,B 0,C 180,E1 -19671.467,E2 -19671.467} C_VEL
LIN {X 0,Y 243.002,Z 282.998,A -85,B 0,C 180,E1 -19672.248,E2 -19672.248} C_VEL
LIN {X 0,Y 246.03,Z 210.48,A -85,B 0,C 180,E1 -19675.001,E2 -19675.001} C_VEL
LIN {X 0,Y 245.023,Z 205.495,A -85,B 0,C 180,E1 -19675.275,E2 -19675.275} C_VEL
LIN {X 0,Y 235.525,Z 176.171,A -85,B 0,C 180,E1 -19677.237,E2 -19677.237} C_VEL
LIN {X 0,Y 234.987,Z 174.341,A -85,B 0,C 180,E1 -19677.427,E2 -19677.427} C_VEL
LIN {X 0,Y 234.896,Z 174.224,A -85,B 0,C 180,E1 -19681.397,E2 -19681.397} C_VEL
LIN {X 0,Y 234.918,Z 174.221,A -85,B 0,C 180,E1 -19685.237,E2 -19685.237} C_VEL
LIN {X 0,Y 234.941,Z 174.218,A -85,B 0,C 180,E1 -19688.962,E2 -19688.962} C_VEL
LIN {X 0,Y 235.054,Z 174.204,A -85,B 0,C 180,E1 -19693.097,E2 -19693.097} C_VEL
LIN {X 0,Y 235.088,Z 174.203,A -85,B 0,C 180,E1 -19697.919,E2 -19697.919} C_VEL
LIN {X 0,Y 235.319,Z 174.171,A -85,B 0,C 180,E1 -19701.411,E2 -19701.411} C_VEL
LIN {X 0,Y 235.356,Z 174.166,A -85,B 0,C 180,E1 -19703.139,E2 -19703.139} C_VEL
LIN {X 0,Y 235.58,Z 174.138,A -85,B 0,C 180,E1 -19708.289,E2 -19708.289} C_VEL
LIN {X 0,Y 235.579,Z 174.14,A -85,B 0,C 180,E1 -19711.708,E2 -19711.708} C_VEL
LIN {X 0,Y 235.349,Z 174.166,A -85,B 0,C 180,E1 -19716.859,E2 -19716.859} C_VEL
LIN {X 0,Y 235.186,Z 174.187,A -85,B 0,C 180,E1 -19720.327,E2 -19720.327} C_VEL
LIN {X 0,Y 235.058,Z 174.204,A -85,B 0,C 180,E1 -19725.609,E2 -19725.609} C_VEL
LIN {X 0,Y 234.959,Z 174.217,A -85,B 0,C 180,E1 -19729.208,E2 -19729.208} C_VEL
LIN {X 0,Y 234.909,Z 174.223,A -85,B 0,C 180,E1 -19732.886,E2 -19732.886} C_VEL
LIN {X 0,Y 234.925,Z 174.219,A -85,B 0,C 180,E1 -19736.661,E2 -19736.661} C_VEL
LIN {X 0,Y 234.898,Z 174.224,A -85,B 0,C 180,E1 -19740.571,E2 -19740.571} C_VEL
LIN {X 0,Y 234.924,Z 174.219,A -85,B 0,C 180,E1 -19744.637,E2 -19744.637} C_VEL
LIN {X 0,Y 234.91,Z 174.225,A -85,B 0,C 180,E1 -19748.933,E2 -19748.933} C_VEL
LIN {X 0,Y 234.85,Z 174.229,A -85,B 0,C 180,E1 -19753.492,E2 -19753.492} C_VEL
LIN {X 0,Y 234.85,Z 174.231,A -85,B 0,C 180,E1 -19756.505,E2 -19756.505} C_VEL
LIN {X 0,Y 234.914,Z 174.222,A -85,B 0,C 180,E1 -19761.077,E2 -19761.077} C_VEL
LIN {X 0,Y 234.921,Z 174.22,A -85,B 0,C 180,E1 -19765.36,E2 -19765.36} C_VEL
LIN {X 0,Y 234.894,Z 174.222,A -85,B 0,C 180,E1 -19769.426,E2 -19769.426} C_VEL
LIN {X 0,Y 234.935,Z 174.219,A -85,B 0,C 180,E1 -19773.819,E2 -19773.819} C_VEL
LIN {X 0,Y 234.93,Z 174.219,A -85,B 0,C 180,E1 -19778.962,E2 -19778.962} C_VEL
LIN {X 0,Y 235.043,Z 174.204,A -85,B 0,C 180,E1 -19783.097,E2 -19783.097} C_VEL
LIN {X 0,Y 235.077,Z 174.202,A -85,B 0,C 180,E1 -19787.92,E2 -19787.92} C_VEL
LIN {X 0,Y 235.309,Z 174.172,A -85,B 0,C 180,E1 -19791.411,E2 -19791.411} C_VEL
LIN {X 0,Y 235.345,Z 174.165,A -85,B 0,C 180,E1 -19793.139,E2 -19793.139} C_VEL
LIN {X 0,Y 235.569,Z 174.141,A -85,B 0,C 180,E1 -19798.29,E2 -19798.29} C_VEL
LIN {X 0,Y 235.569,Z 174.141,A -85,B 0,C 180,E1 -19801.709,E2 -19801.709} C_VEL
LIN {X 0,Y 235.34,Z 174.168,A -85,B 0,C 180,E1 -19806.86,E2 -19806.86} C_VEL
LIN {X 0,Y 235.177,Z 174.186,A -85,B 0,C 180,E1 -19810.329,E2 -19810.329} C_VEL
LIN {X 0,Y 235.05,Z 174.208,A -85,B 0,C 180,E1 -19815.61,E2 -19815.61} C_VEL
LIN {X 0,Y 234.951,Z 174.216,A -85,B 0,C 180,E1 -19819.21,E2 -19819.21} C_VEL
LIN {X 0,Y 234.901,Z 174.223,A -85,B 0,C 180,E1 -19822.889,E2 -19822.889} C_VEL
LIN {X 0,Y 234.919,Z 174.219,A -85,B 0,C 180,E1 -19826.663,E2 -19826.663} C_VEL
LIN {X 0,Y 234.898,Z 174.223,A -85,B 0,C 180,E1 -19830.237,E2 -19830.237} C_VEL
LIN {X 0,Y 234.206,Z 174.311,A -85,B 0,C 180,E1 -19831.667,E2 -19831.667} C_VEL
LIN {X 0,Y 231.343,Z 174.665,A -85,B 0,C 180,E1 -19834,E2 -19834} C_VEL
LIN {X 0,Y 228.932,Z 174.963,A -85,B 0,C 180,E1 -19835.901,E2 -19835.901} C_VEL
LIN {X 0,Y 227.909,Z 175.095,A -85,B 0,C 180,E1 -19837.378,E2 -19837.378} C_VEL
LIN {X 0,Y 227.831,Z 175.101,A -85,B 0,C 180,E1 -19837.878,E2 -19837.878} C_VEL
LIN {X 0,Y 227.78,Z 175.111,A -85,B 0,C 180,E1 -19842.749,E2 -19842.749} C_VEL
LIN {X 0,Y 227.78,Z 175.113,A -85,B 0,C 180,E1 -19847.253,E2 -19847.253} C_VEL
LIN {X 0,Y 227.835,Z 175.103,A -85,B 0,C 180,E1 -19851.909,E2 -19851.909} C_VEL
LIN {X 0,Y 227.951,Z 175.203,A -85,B 0,C 180,E1 -19855.448,E2 -19855.448} C_VEL
LIN {X 0,Y 230.153,Z 186.497,A -85,B 0,C 180,E1 -19860.045,E2 -19860.045} C_VEL
LIN {X 0,Y 230.24,Z 186.965,A -85,B 0,C 180,E1 -19860.231,E2 -19860.231} C_VEL
LIN {X 0,Y 234.916,Z 202.622,A -85,B 0,C 180,E1 -19861.31,E2 -19861.31} C_VEL
LIN {X 0,Y 238.596,Z 235.685,A -85,B 0,C 180,E1 -19862.981,E2 -19862.981} C_VEL
LIN {X 0,Y 235.986,Z 296.086,A -85,B 0,C 180,E1 -19865.36,E2 -19865.36} C_VEL
LIN {X 0,Y 234.896,Z 310.596,A -85,B 0,C 180,E1 -19866.296,E2 -19866.296} C_VEL
LIN {X 0,Y 233.594,Z 322.972,A -85,B 0,C 180,E1 -19867.445,E2 -19867.445} C_VEL
LIN {X 0,Y 232.215,Z 335.113,A -85,B 0,C 180,E1 -19868.939,E2 -19868.939} C_VEL
LIN {X 0,Y 230.748,Z 346.212,A -85,B 0,C 180,E1 -19870.676,E2 -19870.676} C_VEL
LIN {X 0,Y 229.417,Z 356.138,A -85,B 0,C 180,E1 -19872.623,E2 -19872.623} C_VEL
LIN {X 0,Y 228.169,Z 365.27,A -85,B 0,C 180,E1 -19874.824,E2 -19874.824} C_VEL
LIN {X 0,Y 227.166,Z 372.797,A -85,B 0,C 180,E1 -19877.04,E2 -19877.04} C_VEL
LIN {X 0,Y 226.404,Z 380.164,A -85,B 0,C 180,E1 -19879.72,E2 -19879.72} C_VEL
LIN {X 0,Y 226.02,Z 385.109,A -85,B 0,C 180,E1 -19881.958,E2 -19881.958} C_VEL
LIN {X 0,Y 225.823,Z 390.097,A -85,B 0,C 180,E1 -19884.807,E2 -19884.807} C_VEL
LIN {X 0,Y 225.735,Z 392.313,A -85,B 0,C 180,E1 -19886.432,E2 -19886.432} C_VEL
LIN {X 0,Y 225.786,Z 394.308,A -85,B 0,C 180,E1 -19888.218,E2 -19888.218} C_VEL
LIN {X 0,Y 225.783,Z 395.853,A -85,B 0,C 180,E1 -19890.002,E2 -19890.002} C_VEL
LIN {X 0,Y 225.751,Z 396.926,A -85,B 0,C 180,E1 -19891.786,E2 -19891.786} C_VEL
LIN {X 0,Y 225.647,Z 397.802,A -85,B 0,C 180,E1 -19895.363,E2 -19895.363} C_VEL
LIN {X 0,Y 225.831,Z 397.65,A -85,B 0,C 180,E1 -19897.152,E2 -19897.152} C_VEL
LIN {X 0,Y 226.187,Z 397.085,A -85,B 0,C 180,E1 -19898.939,E2 -19898.939} C_VEL
LIN {X 0,Y 227.473,Z 394.731,A -85,B 0,C 180,E1 -19902.492,E2 -19902.492} C_VEL
LIN {X 0,Y 228.933,Z 391.888,A -85,B 0,C 180,E1 -19905.127,E2 -19905.127} C_VEL
LIN {X 0,Y 231.054,Z 388.03,A -85,B 0,C 180,E1 -19907.71,E2 -19907.71} C_VEL
LIN {X 0,Y 233.579,Z 383.113,A -85,B 0,C 180,E1 -19910.245,E2 -19910.245} C_VEL
LIN {X 0,Y 236.867,Z 376.006,A -85,B 0,C 180,E1 -19913.105,E2 -19913.105} C_VEL
LIN {X 0,Y 240.478,Z 368.077,A -85,B 0,C 180,E1 -19915.537,E2 -19915.537} C_VEL
LIN {X 0,Y 244.6,Z 358.401,A -85,B 0,C 180,E1 -19917.835,E2 -19917.835} C_VEL
LIN {X 0,Y 248.346,Z 348.657,A -85,B 0,C 180,E1 -19919.687,E2 -19919.687} C_VEL
LIN {X 0,Y 251.959,Z 337.892,A -85,B 0,C 180,E1 -19921.301,E2 -19921.301} C_VEL
LIN {X 0,Y 255.353,Z 326.042,A -85,B 0,C 180,E1 -19922.694,E2 -19922.694} C_VEL
LIN {X 0,Y 258.437,Z 313.651,A -85,B 0,C 180,E1 -19923.766,E2 -19923.766} C_VEL
LIN {X 0,Y 261.117,Z 299.244,A -85,B 0,C 180,E1 -19924.668,E2 -19924.668} C_VEL
LIN {X 0,Y 263.032,Z 283.332,A -85,B 0,C 180,E1 -19925.335,E2 -19925.335} C_VEL
LIN {X 0,Y 266.805,Z 244.151,A -85,B 0,C 180,E1 -19926.789,E2 -19926.789} C_VEL
LIN {X 0,Y 266.331,Z 239.905,A -85,B 0,C 180,E1 -19927.205,E2 -19927.205} C_VEL
LIN {X 0,Y 263.251,Z 232.075,A -85,B 0,C 180,E1 -19928.704,E2 -19928.704} C_VEL
LIN {X 0,Y 259.141,Z 223.079,A -85,B 0,C 180,E1 -19930.859,E2 -19930.859} C_VEL
LIN {X 0,Y 256.237,Z 217.659,A -85,B 0,C 180,E1 -19932.532,E2 -19932.532} C_VEL
LIN {X 0,Y 253.495,Z 212.789,A -85,B 0,C 180,E1 -19934.265,E2 -19934.265} C_VEL
LIN {X 0,Y 250.389,Z 207.558,A -85,B 0,C 180,E1 -19936.56,E2 -19936.56} C_VEL
LIN {X 0,Y 246.601,Z 201.699,A -85,B 0,C 180,E1 -19940.116,E2 -19940.116} C_VEL
LIN {X 0,Y 243.796,Z 197.649,A -85,B 0,C 180,E1 -19944.287,E2 -19944.287} C_VEL
LIN {X 0,Y 242.824,Z 195.923,A -85,B 0,C 180,E1 -19947.484,E2 -19947.484} C_VEL
LIN {X 0,Y 242.79,Z 195.567,A -85,B 0,C 180,E1 -19950.522,E2 -19950.522} C_VEL
LIN {X 0,Y 243.818,Z 196.784,A -85,B 0,C 180,E1 -19954.024,E2 -19954.024} C_VEL
LIN {X 0,Y 246.736,Z 199.592,A -85,B 0,C 180,E1 -19958.187,E2 -19958.187} C_VEL
LIN {X 0,Y 249.579,Z 203.492,A -85,B 0,C 180,E1 -19960.957,E2 -19960.957} C_VEL
LIN {X 0,Y 250.723,Z 204.951,A -85,B 0,C 180,E1 -19961.886,E2 -19961.886} C_VEL
LIN {X 0,Y 254.071,Z 209.8,A -85,B 0,C 180,E1 -19964.278,E2 -19964.278} C_VEL
LIN {X 0,Y 257.334,Z 214.69,A -85,B 0,C 180,E1 -19966.232,E2 -19966.232} C_VEL
LIN {X 0,Y 261.005,Z 220.838,A -85,B 0,C 180,E1 -19968.206,E2 -19968.206} C_VEL
LIN {X 0,Y 266.661,Z 232.29,A -85,B 0,C 180,E1 -19970.935,E2 -19970.935} C_VEL
LIN {X 0,Y 267.577,Z 234.563,A -85,B 0,C 180,E1 -19971.358,E2 -19971.358} C_VEL
LIN {X 0,Y 262.296,Z 286.502,A -85,B 0,C 180,E1 -19973.298,E2 -19973.298} C_VEL
LIN {X 0,Y 260.103,Z 300.202,A -85,B 0,C 180,E1 -19974.088,E2 -19974.088} C_VEL
LIN {X 0,Y 257.589,Z 312.464,A -85,B 0,C 180,E1 -19975.109,E2 -19975.109} C_VEL
LIN {X 0,Y 254.558,Z 324.188,A -85,B 0,C 180,E1 -19976.383,E2 -19976.383} C_VEL
LIN {X 0,Y 251.095,Z 335.423,A -85,B 0,C 180,E1 -19977.955,E2 -19977.955} C_VEL
LIN {X 0,Y 246.988,Z 346.715,A -85,B 0,C 180,E1 -19980,E2 -19980} C_VEL
LIN {X 0,Y 243.293,Z 355.709,A -85,B 0,C 180,E1 -19982.07,E2 -19982.07} C_VEL
LIN {X 0,Y 239.37,Z 364.286,A -85,B 0,C 180,E1 -19984.594,E2 -19984.594} C_VEL
LIN {X 0,Y 236.437,Z 370.238,A -85,B 0,C 180,E1 -19986.829,E2 -19986.829} C_VEL
LIN {X 0,Y 233.43,Z 375.866,A -85,B 0,C 180,E1 -19989.532,E2 -19989.532} C_VEL
LIN {X 0,Y 230.55,Z 380.719,A -85,B 0,C 180,E1 -19992.71,E2 -19992.71} C_VEL
LIN {X 0,Y 228.342,Z 384.089,A -85,B 0,C 180,E1 -19996.082,E2 -19996.082} C_VEL
LIN {X 0,Y 227.417,Z 385.308,A -85,B 0,C 180,E1 -19998.002,E2 -19998.002} C_VEL
LIN {X 0,Y 226.239,Z 386.224,A -85,B 0,C 180,E1 -20001.258,E2 -20001.258} C_VEL
LIN {X 0,Y 225.627,Z 386.004,A -85,B 0,C 180,E1 -20003.888,E2 -20003.888} C_VEL
LIN {X 0,Y 225.331,Z 385.217,A -85,B 0,C 180,E1 -20005.891,E2 -20005.891} C_VEL
LIN {X 0,Y 225.261,Z 382.883,A -85,B 0,C 180,E1 -20009.12,E2 -20009.12} C_VEL
LIN {X 0,Y 225.523,Z 379.59,A -85,B 0,C 180,E1 -20011.991,E2 -20011.991} C_VEL
LIN {X 0,Y 225.837,Z 376.402,A -85,B 0,C 180,E1 -20014.067,E2 -20014.067} C_VEL
LIN {X 0,Y 226.44,Z 370.166,A -85,B 0,C 180,E1 -20017.246,E2 -20017.246} C_VEL
LIN {X 0,Y 227.171,Z 363.652,A -85,B 0,C 180,E1 -20019.813,E2 -20019.813} C_VEL
LIN {X 0,Y 228.231,Z 355.669,A -85,B 0,C 180,E1 -20022.348,E2 -20022.348} C_VEL
LIN {X 0,Y 229.486,Z 346.2,A -85,B 0,C 180,E1 -20024.78,E2 -20024.78} C_VEL
LIN {X 0,Y 230.88,Z 335.638,A -85,B 0,C 180,E1 -20026.934,E2 -20026.934} C_VEL
LIN {X 0,Y 232.367,Z 324.15,A -85,B 0,C 180,E1 -20028.807,E2 -20028.807} C_VEL
LIN {X 0,Y 233.855,Z 311.821,A -85,B 0,C 180,E1 -20030.364,E2 -20030.364} C_VEL
LIN {X 0,Y 234.95,Z 299.407,A -85,B 0,C 180,E1 -20031.569,E2 -20031.569} C_VEL
LIN {X 0,Y 235.882,Z 286.084,A -85,B 0,C 180,E1 -20032.494,E2 -20032.494} C_VEL
LIN {X 0,Y 236.793,Z 267.513,A -85,B 0,C 180,E1 -20033.294,E2 -20033.294} C_VEL
LIN {X 0,Y 239.237,Z 211.323,A -85,B 0,C 180,E1 -20035.457,E2 -20035.457} C_VEL
LIN {X 0,Y 238.048,Z 206.27,A -85,B 0,C 180,E1 -20035.758,E2 -20035.758} C_VEL
LIN {X 0,Y 228.794,Z 177.701,A -85,B 0,C 180,E1 -20037.741,E2 -20037.741} C_VEL
LIN {X 0,Y 227.918,Z 175.094,A -85,B 0,C 180,E1 -20037.961,E2 -20037.961} C_VEL
LIN {X 0,Y 227.838,Z 175.107,A -85,B 0,C 180,E1 -20042.437,E2 -20042.437} C_VEL
LIN {X 0,Y 227.87,Z 175.102,A -85,B 0,C 180,E1 -20046.361,E2 -20046.361} C_VEL
LIN {X 0,Y 227.893,Z 175.1,A -85,B 0,C 180,E1 -20050.169,E2 -20050.169} C_VEL
LIN {X 0,Y 228.013,Z 175.084,A -85,B 0,C 180,E1 -20053.893,E2 -20053.893} C_VEL
LIN {X 0,Y 228.129,Z 175.067,A -85,B 0,C 180,E1 -20059.347,E2 -20059.347} C_VEL
LIN {X 0,Y 228.308,Z 175.044,A -85,B 0,C 180,E1 -20062.926,E2 -20062.926} C_VEL
LIN {X 0,Y 228.538,Z 175.015,A -85,B 0,C 180,E1 -20068.236,E2 -20068.236} C_VEL
LIN {X 0,Y 228.537,Z 175.017,A -85,B 0,C 180,E1 -20071.761,E2 -20071.761} C_VEL
LIN {X 0,Y 228.301,Z 175.044,A -85,B 0,C 180,E1 -20077.072,E2 -20077.072} C_VEL
LIN {X 0,Y 228.127,Z 175.066,A -85,B 0,C 180,E1 -20080.65,E2 -20080.65} C_VEL
LIN {X 0,Y 228.009,Z 175.079,A -85,B 0,C 180,E1 -20086.104,E2 -20086.104} C_VEL
LIN {X 0,Y 227.919,Z 175.094,A -85,B 0,C 180,E1 -20091.715,E2 -20091.715} C_VEL
LIN {X 0,Y 227.903,Z 175.093,A -85,B 0,C 180,E1 -20096.581,E2 -20096.581} C_VEL
LIN {X 0,Y 227.873,Z 175.098,A -85,B 0,C 180,E1 -20100.279,E2 -20100.279} C_VEL
LIN {X 0,Y 227.875,Z 175.096,A -85,B 0,C 180,E1 -20103.719,E2 -20103.719} C_VEL
LIN {X 0,Y 227.838,Z 175.103,A -85,B 0,C 180,E1 -20108.09,E2 -20108.09} C_VEL
LIN {X 0,Y 227.783,Z 175.109,A -85,B 0,C 180,E1 -20112.747,E2 -20112.747} C_VEL
LIN {X 0,Y 227.782,Z 175.11,A -85,B 0,C 180,E1 -20117.25,E2 -20117.25} C_VEL
LIN {X 0,Y 227.836,Z 175.101,A -85,B 0,C 180,E1 -20121.907,E2 -20121.907} C_VEL
LIN {X 0,Y 227.874,Z 175.1,A -85,B 0,C 180,E1 -20126.376,E2 -20126.376} C_VEL
LIN {X 0,Y 227.871,Z 175.1,A -85,B 0,C 180,E1 -20130.43,E2 -20130.43} C_VEL
LIN {X 0,Y 227.866,Z 175.102,A -85,B 0,C 180,E1 -20134.418,E2 -20134.418} C_VEL
LIN {X 0,Y 227.913,Z 175.094,A -85,B 0,C 180,E1 -20138.282,E2 -20138.282} C_VEL
LIN {X 0,Y 228.002,Z 175.083,A -85,B 0,C 180,E1 -20143.893,E2 -20143.893} C_VEL
LIN {X 0,Y 228.118,Z 175.068,A -85,B 0,C 180,E1 -20149.347,E2 -20149.347} C_VEL
LIN {X 0,Y 228.298,Z 175.043,A -85,B 0,C 180,E1 -20152.926,E2 -20152.926} C_VEL
LIN {X 0,Y 228.527,Z 175.019,A -85,B 0,C 180,E1 -20158.237,E2 -20158.237} C_VEL
LIN {X 0,Y 228.527,Z 175.018,A -85,B 0,C 180,E1 -20161.762,E2 -20161.762} C_VEL
LIN {X 0,Y 228.292,Z 175.046,A -85,B 0,C 180,E1 -20167.073,E2 -20167.073} C_VEL
LIN {X 0,Y 228.118,Z 175.065,A -85,B 0,C 180,E1 -20170.652,E2 -20170.652} C_VEL
LIN {X 0,Y 228.001,Z 175.083,A -85,B 0,C 180,E1 -20176.106,E2 -20176.106} C_VEL
LIN {X 0,Y 227.912,Z 175.096,A -85,B 0,C 180,E1 -20181.718,E2 -20181.718} C_VEL
LIN {X 0,Y 227.896,Z 175.093,A -85,B 0,C 180,E1 -20186.583,E2 -20186.583} C_VEL
LIN {X 0,Y 227.867,Z 175.099,A -85,B 0,C 180,E1 -20190.281,E2 -20190.281} C_VEL
LIN {X 0,Y 227.87,Z 175.098,A -85,B 0,C 180,E1 -20193.721,E2 -20193.721} C_VEL
LIN {X 0,Y 227.831,Z 175.101,A -85,B 0,C 180,E1 -20197.878,E2 -20197.878} C_VEL
LIN {X 0,Y 227.181,Z 175.189,A -85,B 0,C 180,E1 -20199.354,E2 -20199.354} C_VEL
LIN {X 0,Y 224.346,Z 175.548,A -85,B 0,C 180,E1 -20201.762,E2 -20201.762} C_VEL
LIN {X 0,Y 221.081,Z 175.949,A -85,B 0,C 180,E1 -20204.738,E2 -20204.738} C_VEL
LIN {X 0,Y 220.736,Z 175.988,A -85,B 0,C 180,E1 -20205.769,E2 -20205.769} C_VEL
LIN {X 0,Y 220.777,Z 175.984,A -85,B 0,C 180,E1 -20210.459,E2 -20210.459} C_VEL
LIN {X 0,Y 220.881,Z 175.98,A -85,B 0,C 180,E1 -20215.062,E2 -20215.062} C_VEL
LIN {X 0,Y 223.077,Z 187.065,A -85,B 0,C 180,E1 -20219.649,E2 -20219.649} C_VEL
LIN {X 0,Y 228.335,Z 204.941,A -85,B 0,C 180,E1 -20220.885,E2 -20220.885} C_VEL
LIN {X 0,Y 231.771,Z 236.272,A -85,B 0,C 180,E1 -20222.515,E2 -20222.515} C_VEL
LIN {X 0,Y 229.116,Z 295.745,A -85,B 0,C 180,E1 -20224.934,E2 -20224.934} C_VEL
LIN {X 0,Y 227.996,Z 310.217,A -85,B 0,C 180,E1 -20225.895,E2 -20225.895} C_VEL
LIN {X 0,Y 226.793,Z 321.65,A -85,B 0,C 180,E1 -20226.971,E2 -20226.971} C_VEL
LIN {X 0,Y 225.365,Z 333.964,A -85,B 0,C 180,E1 -20228.507,E2 -20228.507} C_VEL
LIN {X 0,Y 223.949,Z 344.391,A -85,B 0,C 180,E1 -20230.15,E2 -20230.15} C_VEL
LIN {X 0,Y 222.444,Z 355.284,A -85,B 0,C 180,E1 -20232.298,E2 -20232.298} C_VEL
LIN {X 0,Y 221.069,Z 365.339,A -85,B 0,C 180,E1 -20234.797,E2 -20234.797} C_VEL
LIN {X 0,Y 220.036,Z 372.799,A -85,B 0,C 180,E1 -20237.082,E2 -20237.082} C_VEL
LIN {X 0,Y 219.288,Z 380.119,A -85,B 0,C 180,E1 -20239.849,E2 -20239.849} C_VEL
LIN {X 0,Y 218.873,Z 385.9,A -85,B 0,C 180,E1 -20242.622,E2 -20242.622} C_VEL
LIN {X 0,Y 218.735,Z 389.7,A -85,B 0,C 180,E1 -20244.897,E2 -20244.897} C_VEL
LIN {X 0,Y 218.721,Z 393.72,A -85,B 0,C 180,E1 -20248.16,E2 -20248.16} C_VEL
LIN {X 0,Y 218.718,Z 395.339,A -85,B 0,C 180,E1 -20250.002,E2 -20250.002} C_VEL
LIN {X 0,Y 218.68,Z 396.525,A -85,B 0,C 180,E1 -20251.843,E2 -20251.843} C_VEL
LIN {X 0,Y 218.52,Z 397.413,A -85,B 0,C 180,E1 -20254.427,E2 -20254.427} C_VEL
LIN {X 0,Y 218.788,Z 397.482,A -85,B 0,C 180,E1 -20257.384,E2 -20257.384} C_VEL
LIN {X 0,Y 219.765,Z 396.157,A -85,B 0,C 180,E1 -20261.064,E2 -20261.064} C_VEL
LIN {X 0,Y 221.495,Z 393.164,A -85,B 0,C 180,E1 -20264.706,E2 -20264.706} C_VEL
LIN {X 0,Y 223.482,Z 389.845,A -85,B 0,C 180,E1 -20267.384,E2 -20267.384} C_VEL
LIN {X 0,Y 226.073,Z 385.483,A -85,B 0,C 180,E1 -20269.998,E2 -20269.998} C_VEL
LIN {X 0,Y 229.515,Z 378.813,A -85,B 0,C 180,E1 -20273.058,E2 -20273.058} C_VEL
LIN {X 0,Y 233.545,Z 370.635,A -85,B 0,C 180,E1 -20275.872,E2 -20275.872} C_VEL
LIN {X 0,Y 237.739,Z 361.741,A -85,B 0,C 180,E1 -20278.23,E2 -20278.23} C_VEL
LIN {X 0,Y 241.956,Z 351.703,A -85,B 0,C 180,E1 -20280.312,E2 -20280.312} C_VEL
LIN {X 0,Y 246.097,Z 340.417,A -85,B 0,C 180,E1 -20282.135,E2 -20282.135} C_VEL
LIN {X 0,Y 250.063,Z 327.74,A -85,B 0,C 180,E1 -20283.717,E2 -20283.717} C_VEL
LIN {X 0,Y 253.49,Z 315.017,A -85,B 0,C 180,E1 -20284.879,E2 -20284.879} C_VEL
LIN {X 0,Y 256.301,Z 301.601,A -85,B 0,C 180,E1 -20285.763,E2 -20285.763} C_VEL
LIN {X 0,Y 258.32,Z 287.556,A -85,B 0,C 180,E1 -20286.403,E2 -20286.403} C_VEL
LIN {X 0,Y 262.47,Z 245.745,A -85,B 0,C 180,E1 -20287.982,E2 -20287.982} C_VEL
LIN {X 0,Y 262.132,Z 243.343,A -85,B 0,C 180,E1 -20288.257,E2 -20288.257} C_VEL
LIN {X 0,Y 259.358,Z 235.891,A -85,B 0,C 180,E1 -20289.77,E2 -20289.77} C_VEL
LIN {X 0,Y 255.632,Z 227.687,A -85,B 0,C 180,E1 -20291.887,E2 -20291.887} C_VEL
LIN {X 0,Y 253.29,Z 223.111,A -85,B 0,C 180,E1 -20293.344,E2 -20293.344} C_VEL
LIN {X 0,Y 251.043,Z 218.845,A -85,B 0,C 180,E1 -20294.907,E2 -20294.907} C_VEL
LIN {X 0,Y 248.243,Z 213.93,A -85,B 0,C 180,E1 -20297.105,E2 -20297.105} C_VEL
LIN {X 0,Y 244.919,Z 208.396,A -85,B 0,C 180,E1 -20300.496,E2 -20300.496} C_VEL
LIN {X 0,Y 242.357,Z 204.505,A -85,B 0,C 180,E1 -20304.552,E2 -20304.552} C_VEL
LIN {X 0,Y 241.51,Z 202.876,A -85,B 0,C 180,E1 -20307.557,E2 -20307.557} C_VEL
LIN {X 0,Y 241.529,Z 202.578,A -85,B 0,C 180,E1 -20310.804,E2 -20310.804} C_VEL
LIN {X 0,Y 242.789,Z 204.124,A -85,B 0,C 180,E1 -20314.613,E2 -20314.613} C_VEL
LIN {X 0,Y 245.04,Z 206.314,A -85,B 0,C 180,E1 -20317.787,E2 -20317.787} C_VEL
LIN {X 0,Y 247.856,Z 210.278,A -85,B 0,C 180,E1 -20320.686,E2 -20320.686} C_VEL
LIN {X 0,Y 249.82,Z 213.258,A -85,B 0,C 180,E1 -20322.332,E2 -20322.332} C_VEL
LIN {X 0,Y 251.92,Z 216.348,A -85,B 0,C 180,E1 -20323.848,E2 -20323.848} C_VEL
LIN {X 0,Y 254.782,Z 220.873,A -85,B 0,C 180,E1 -20325.675,E2 -20325.675} C_VEL
LIN {X 0,Y 257.957,Z 226.488,A -85,B 0,C 180,E1 -20327.526,E2 -20327.526} C_VEL
LIN {X 0,Y 263.151,Z 237.554,A -85,B 0,C 180,E1 -20330.215,E2 -20330.215} C_VEL
LIN {X 0,Y 257.922,Z 286.791,A -85,B 0,C 180,E1 -20332.069,E2 -20332.069} C_VEL
LIN {X 0,Y 255.714,Z 300.006,A -85,B 0,C 180,E1 -20332.83,E2 -20332.83} C_VEL
LIN {X 0,Y 253.151,Z 311.972,A -85,B 0,C 180,E1 -20333.825,E2 -20333.825} C_VEL
LIN {X 0,Y 250.215,Z 322.707,A -85,B 0,C 180,E1 -20334.965,E2 -20334.965} C_VEL
LIN {X 0,Y 246.183,Z 335.373,A -85,B 0,C 180,E1 -20336.727,E2 -20336.727} C_VEL
LIN {X 0,Y 241.899,Z 346.575,A -85,B 0,C 180,E1 -20338.752,E2 -20338.752} C_VEL
LIN {X 0,Y 237.99,Z 355.65,A -85,B 0,C 180,E1 -20340.853,E2 -20340.853} C_VEL
LIN {X 0,Y 233.644,Z 364.378,A -85,B 0,C 180,E1 -20343.449,E2 -20343.449} C_VEL
LIN {X 0,Y 230.022,Z 371.298,A -85,B 0,C 180,E1 -20346.139,E2 -20346.139} C_VEL
LIN {X 0,Y 226.837,Z 376.764,A -85,B 0,C 180,E1 -20348.912,E2 -20348.912} C_VEL
LIN {X 0,Y 224.139,Z 380.902,A -85,B 0,C 180,E1 -20351.76,E2 -20351.76} C_VEL
LIN {X 0,Y 222.043,Z 383.837,A -85,B 0,C 180,E1 -20354.668,E2 -20354.668} C_VEL
LIN {X 0,Y 220.69,Z 385.493,A -85,B 0,C 180,E1 -20357.178,E2 -20357.178} C_VEL
LIN {X 0,Y 219.321,Z 386.449,A -85,B 0,C 180,E1 -20360.64,E2 -20360.64} C_VEL
LIN {X 0,Y 218.766,Z 386.354,A -85,B 0,C 180,E1 -20362.676,E2 -20362.676} C_VEL
LIN {X 0,Y 218.265,Z 385.331,A -85,B 0,C 180,E1 -20365.63,E2 -20365.63} C_VEL
LIN {X 0,Y 218.199,Z 382.293,A -85,B 0,C 180,E1 -20369.58,E2 -20369.58} C_VEL
LIN {X 0,Y 218.604,Z 377.815,A -85,B 0,C 180,E1 -20373.131,E2 -20373.131} C_VEL
LIN {X 0,Y 219.044,Z 372.743,A -85,B 0,C 180,E1 -20376.017,E2 -20376.017} C_VEL
LIN {X 0,Y 219.869,Z 365.598,A -85,B 0,C 180,E1 -20379.147,E2 -20379.147} C_VEL
LIN {X 0,Y 220.905,Z 357.549,A -85,B 0,C 180,E1 -20381.922,E2 -20381.922} C_VEL
LIN {X 0,Y 222.151,Z 348.438,A -85,B 0,C 180,E1 -20384.424,E2 -20384.424} C_VEL
LIN {X 0,Y 223.467,Z 338.396,A -85,B 0,C 180,E1 -20386.66,E2 -20386.66} C_VEL
LIN {X 0,Y 224.945,Z 327.627,A -85,B 0,C 180,E1 -20388.577,E2 -20388.577} C_VEL
LIN {X 0,Y 226.466,Z 315.335,A -85,B 0,C 180,E1 -20390.304,E2 -20390.304} C_VEL
LIN {X 0,Y 227.789,Z 302.556,A -85,B 0,C 180,E1 -20391.676,E2 -20391.676} C_VEL
LIN {X 0,Y 228.832,Z 288.188,A -85,B 0,C 180,E1 -20392.786,E2 -20392.786} C_VEL
LIN {X 0,Y 229.708,Z 273.97,A -85,B 0,C 180,E1 -20393.477,E2 -20393.477} C_VEL
LIN {X 0,Y 232.493,Z 212.346,A -85,B 0,C 180,E1 -20395.929,E2 -20395.929} C_VEL
LIN {X 0,Y 227.325,Z 195.035,A -85,B 0,C 180,E1 -20397.096,E2 -20397.096} C_VEL
LIN {X 0,Y 221.672,Z 178.548,A -85,B 0,C 180,E1 -20398.324,E2 -20398.324} C_VEL
LIN {X 0,Y 220.839,Z 175.977,A -85,B 0,C 180,E1 -20398.545,E2 -20398.545} C_VEL
LIN {X 0,Y 220.834,Z 175.976,A -85,B 0,C 180,E1 -20403.54,E2 -20403.54} C_VEL
LIN {X 0,Y 220.859,Z 175.973,A -85,B 0,C 180,E1 -20407.55,E2 -20407.55} C_VEL
LIN {X 0,Y 220.92,Z 175.966,A -85,B 0,C 180,E1 -20412.628,E2 -20412.628} C_VEL
LIN {X 0,Y 220.979,Z 175.958,A -85,B 0,C 180,E1 -20417.135,E2 -20417.135} C_VEL
LIN {X 0,Y 221.198,Z 175.93,A -85,B 0,C 180,E1 -20420.858,E2 -20420.858} C_VEL
LIN {X 0,Y 221.246,Z 175.924,A -85,B 0,C 180,E1 -20422.699,E2 -20422.699} C_VEL
LIN {X 0,Y 221.471,Z 175.896,A -85,B 0,C 180,E1 -20428.18,E2 -20428.18} C_VEL
LIN {X 0,Y 221.471,Z 175.898,A -85,B 0,C 180,E1 -20431.817,E2 -20431.817} C_VEL
LIN {X 0,Y 221.238,Z 175.925,A -85,B 0,C 180,E1 -20437.299,E2 -20437.299} C_VEL
LIN {X 0,Y 221.052,Z 175.948,A -85,B 0,C 180,E1 -20440.996,E2 -20440.996} C_VEL
LIN {X 0,Y 220.971,Z 175.955,A -85,B 0,C 180,E1 -20446.632,E2 -20446.632} C_VEL
LIN {X 0,Y 220.846,Z 175.974,A -85,B 0,C 180,E1 -20450.489,E2 -20450.489} C_VEL
LIN {X 0,Y 220.796,Z 175.978,A -85,B 0,C 180,E1 -20454.441,E2 -20454.441} C_VEL
LIN {X 0,Y 220.799,Z 175.98,A -85,B 0,C 180,E1 -20458.517,E2 -20458.517} C_VEL
LIN {X 0,Y 220.811,Z 175.978,A -85,B 0,C 180,E1 -20462.755,E2 -20462.755} C_VEL
LIN {X 0,Y 220.8,Z 175.982,A -85,B 0,C 180,E1 -20467.273,E2 -20467.273} C_VEL
LIN {X 0,Y 220.745,Z 175.982,A -85,B 0,C 180,E1 -20471.956,E2 -20471.956} C_VEL
LIN {X 0,Y 220.75,Z 175.986,A -85,B 0,C 180,E1 -20475.539,E2 -20475.539} C_VEL
LIN {X 0,Y 220.777,Z 175.981,A -85,B 0,C 180,E1 -20480.456,E2 -20480.456} C_VEL
LIN {X 0,Y 220.821,Z 175.98,A -85,B 0,C 180,E1 -20482.791,E2 -20482.791} C_VEL
LIN {X 0,Y 220.808,Z 175.977,A -85,B 0,C 180,E1 -20487.242,E2 -20487.242} C_VEL
LIN {X 0,Y 220.794,Z 175.98,A -85,B 0,C 180,E1 -20491.48,E2 -20491.48} C_VEL
LIN {X 0,Y 220.797,Z 175.978,A -85,B 0,C 180,E1 -20495.556,E2 -20495.556} C_VEL
LIN {X 0,Y 220.84,Z 175.974,A -85,B 0,C 180,E1 -20499.508,E2 -20499.508} C_VEL
LIN {X 0,Y 220.964,Z 175.958,A -85,B 0,C 180,E1 -20503.366,E2 -20503.366} C_VEL
LIN {X 0,Y 221.043,Z 175.949,A -85,B 0,C 180,E1 -20509.002,E2 -20509.002} C_VEL
LIN {X 0,Y 221.235,Z 175.923,A -85,B 0,C 180,E1 -20512.699,E2 -20512.699} C_VEL
LIN {X 0,Y 221.461,Z 175.899,A -85,B 0,C 180,E1 -20518.181,E2 -20518.181} C_VEL
LIN {X 0,Y 221.46,Z 175.897,A -85,B 0,C 180,E1 -20521.818,E2 -20521.818} C_VEL
LIN {X 0,Y 221.229,Z 175.927,A -85,B 0,C 180,E1 -20527.3,E2 -20527.3} C_VEL
LIN {X 0,Y 221.043,Z 175.946,A -85,B 0,C 180,E1 -20530.997,E2 -20530.997} C_VEL
LIN {X 0,Y 220.963,Z 175.958,A -85,B 0,C 180,E1 -20536.634,E2 -20536.634} C_VEL
LIN {X 0,Y 220.839,Z 175.973,A -85,B 0,C 180,E1 -20540.491,E2 -20540.491} C_VEL
LIN {X 0,Y 220.789,Z 175.98,A -85,B 0,C 180,E1 -20544.444,E2 -20544.444} C_VEL
LIN {X 0,Y 220.793,Z 175.978,A -85,B 0,C 180,E1 -20548.519,E2 -20548.519} C_VEL
LIN {X 0,Y 220.806,Z 175.979,A -85,B 0,C 180,E1 -20552.758,E2 -20552.758} C_VEL
LIN {X 0,Y 220.796,Z 175.98,A -85,B 0,C 180,E1 -20557.276,E2 -20557.276} C_VEL
LIN {X 0,Y 220.742,Z 175.985,A -85,B 0,C 180,E1 -20561.959,E2 -20561.959} C_VEL
LIN {X 0,Y 220.736,Z 175.988,A -85,B 0,C 180,E1 -20565.769,E2 -20565.769} C_VEL
LIN {X 0,Y 220.035,Z 176.077,A -85,B 0,C 180,E1 -20567.291,E2 -20567.291} C_VEL
LIN {X 0,Y 217.201,Z 176.428,A -85,B 0,C 180,E1 -20569.778,E2 -20569.778} C_VEL
LIN {X 0,Y 214.834,Z 176.723,A -85,B 0,C 180,E1 -20571.808,E2 -20571.808} C_VEL
LIN {X 0,Y 213.85,Z 176.847,A -85,B 0,C 180,E1 -20573.384,E2 -20573.384} C_VEL
LIN {X 0,Y 213.784,Z 176.853,A -85,B 0,C 180,E1 -20573.917,E2 -20573.917} C_VEL
LIN {X 0,Y 213.857,Z 176.995,A -85,B 0,C 180,E1 -20574.766,E2 -20574.766} C_VEL
LIN {X 0,Y 215.788,Z 186.844,A -85,B 0,C 180,E1 -20578.991,E2 -20578.991} C_VEL
LIN {X 0,Y 221.619,Z 206.385,A -85,B 0,C 180,E1 -20580.413,E2 -20580.413} C_VEL
LIN {X 0,Y 224.9,Z 236.983,A -85,B 0,C 180,E1 -20582.049,E2 -20582.049} C_VEL
LIN {X 0,Y 222.202,Z 295.695,A -85,B 0,C 180,E1 -20584.537,E2 -20584.537} C_VEL
LIN {X 0,Y 221.121,Z 309.405,A -85,B 0,C 180,E1 -20585.472,E2 -20585.472} C_VEL
LIN {X 0,Y 219.77,Z 321.979,A -85,B 0,C 180,E1 -20586.69,E2 -20586.69} C_VEL
LIN {X 0,Y 218.317,Z 334.192,A -85,B 0,C 180,E1 -20588.274,E2 -20588.274} C_VEL
LIN {X 0,Y 216.789,Z 345.147,A -85,B 0,C 180,E1 -20590.075,E2 -20590.075} C_VEL
LIN {X 0,Y 215.478,Z 354.357,A -85,B 0,C 180,E1 -20591.952,E2 -20591.952} C_VEL
LIN {X 0,Y 214.179,Z 363.705,A -85,B 0,C 180,E1 -20594.295,E2 -20594.295} C_VEL
LIN {X 0,Y 212.937,Z 372.806,A -85,B 0,C 180,E1 -20597.129,E2 -20597.129} C_VEL
LIN {X 0,Y 212.19,Z 380.074,A -85,B 0,C 180,E1 -20599.988,E2 -20599.988} C_VEL
LIN {X 0,Y 211.823,Z 384.983,A -85,B 0,C 180,E1 -20602.375,E2 -20602.375} C_VEL
LIN {X 0,Y 211.676,Z 389.16,A -85,B 0,C 180,E1 -20604.906,E2 -20604.906} C_VEL
LIN {X 0,Y 211.655,Z 393.119,A -85,B 0,C 180,E1 -20608.099,E2 -20608.099} C_VEL
LIN {X 0,Y 211.655,Z 394.804,A -85,B 0,C 180,E1 -20610.002,E2 -20610.002} C_VEL
LIN {X 0,Y 211.609,Z 396.056,A -85,B 0,C 180,E1 -20611.905,E2 -20611.905} C_VEL
LIN {X 0,Y 211.419,Z 397.021,A -85,B 0,C 180,E1 -20614.244,E2 -20614.244} C_VEL
LIN {X 0,Y 211.721,Z 397.314,A -85,B 0,C 180,E1 -20617.632,E2 -20617.632} C_VEL
LIN {X 0,Y 212.784,Z 396.156,A -85,B 0,C 180,E1 -20621.432,E2 -20621.432} C_VEL
LIN {X 0,Y 213.619,Z 395.003,A -85,B 0,C 180,E1 -20623.316,E2 -20623.316} C_VEL
LIN {X 0,Y 215.257,Z 392.478,A -85,B 0,C 180,E1 -20626.114,E2 -20626.114} C_VEL
LIN {X 0,Y 217.609,Z 388.979,A -85,B 0,C 180,E1 -20628.844,E2 -20628.844} C_VEL
LIN {X 0,Y 220.381,Z 384.436,A -85,B 0,C 180,E1 -20631.516,E2 -20631.516} C_VEL
LIN {X 0,Y 224.006,Z 377.881,A -85,B 0,C 180,E1 -20634.516,E2 -20634.516} C_VEL
LIN {X 0,Y 227.95,Z 370.542,A -85,B 0,C 180,E1 -20637.051,E2 -20637.051} C_VEL
LIN {X 0,Y 232.398,Z 361.648,A -85,B 0,C 180,E1 -20639.436,E2 -20639.436} C_VEL
LIN {X 0,Y 236.857,Z 351.688,A -85,B 0,C 180,E1 -20641.533,E2 -20641.533} C_VEL
LIN {X 0,Y 241.215,Z 340.569,A -85,B 0,C 180,E1 -20643.364,E2 -20643.364} C_VEL
LIN {X 0,Y 244.89,Z 329.646,A -85,B 0,C 180,E1 -20644.779,E2 -20644.779} C_VEL
LIN {X 0,Y 248.672,Z 316.487,A -85,B 0,C 180,E1 -20646.031,E2 -20646.031} C_VEL
LIN {X 0,Y 251.594,Z 303.756,A -85,B 0,C 180,E1 -20646.913,E2 -20646.913} C_VEL
LIN {X 0,Y 253.766,Z 290.166,A -85,B 0,C 180,E1 -20647.585,E2 -20647.585} C_VEL
LIN {X 0,Y 258.402,Z 247.541,A -85,B 0,C 180,E1 -20649.221,E2 -20649.221} C_VEL
LIN {X 0,Y 255.997,Z 240.928,A -85,B 0,C 180,E1 -20650.606,E2 -20650.606} C_VEL
LIN {X 0,Y 252.674,Z 233.123,A -85,B 0,C 180,E1 -20652.679,E2 -20652.679} C_VEL
LIN {X 0,Y 250.671,Z 229.018,A -85,B 0,C 180,E1 -20654.01,E2 -20654.01} C_VEL
LIN {X 0,Y 248.659,Z 224.978,A -85,B 0,C 180,E1 -20655.534,E2 -20655.534} C_VEL
LIN {X 0,Y 246.195,Z 220.346,A -85,B 0,C 180,E1 -20657.633,E2 -20657.633} C_VEL
LIN {X 0,Y 243.191,Z 215.013,A -85,B 0,C 180,E1 -20660.928,E2 -20660.928} C_VEL
LIN {X 0,Y 240.878,Z 211.297,A -85,B 0,C 180,E1 -20664.904,E2 -20664.904} C_VEL
LIN {X 0,Y 240.115,Z 209.71,A -85,B 0,C 180,E1 -20668.208,E2 -20668.208} C_VEL
LIN {X 0,Y 240.302,Z 209.67,A -85,B 0,C 180,E1 -20671.332,E2 -20671.332} C_VEL
LIN {X 0,Y 241.747,Z 211.495,A -85,B 0,C 180,E1 -20675.192,E2 -20675.192} C_VEL
LIN {X 0,Y 243.381,Z 213.054,A -85,B 0,C 180,E1 -20677.441,E2 -20677.441} C_VEL
LIN {X 0,Y 245.9,Z 216.81,A -85,B 0,C 180,E1 -20680.21,E2 -20680.21} C_VEL
LIN {X 0,Y 247.237,Z 219.014,A -85,B 0,C 180,E1 -20681.463,E2 -20681.463} C_VEL
LIN {X 0,Y 249.661,Z 222.654,A -85,B 0,C 180,E1 -20683.316,E2 -20683.316} C_VEL
LIN {X 0,Y 252.168,Z 226.898,A -85,B 0,C 180,E1 -20685.061,E2 -20685.061} C_VEL
LIN {X 0,Y 255.227,Z 232.573,A -85,B 0,C 180,E1 -20686.928,E2 -20686.928} C_VEL
LIN {X 0,Y 258.967,Z 240.781,A -85,B 0,C 180,E1 -20689.02,E2 -20689.02} C_VEL
LIN {X 0,Y 253.742,Z 286.87,A -85,B 0,C 180,E1 -20690.786,E2 -20690.786} C_VEL
LIN {X 0,Y 251.355,Z 300.327,A -85,B 0,C 180,E1 -20691.559,E2 -20691.559} C_VEL
LIN {X 0,Y 248.504,Z 312.94,A -85,B 0,C 180,E1 -20692.62,E2 -20692.62} C_VEL
LIN {X 0,Y 245.277,Z 324.097,A -85,B 0,C 180,E1 -20693.832,E2 -20693.832} C_VEL
LIN {X 0,Y 241.74,Z 334.603,A -85,B 0,C 180,E1 -20695.307,E2 -20695.307} C_VEL
LIN {X 0,Y 237.431,Z 345.439,A -85,B 0,C 180,E1 -20697.243,E2 -20697.243} C_VEL
LIN {X 0,Y 233.017,Z 355.116,A -85,B 0,C 180,E1 -20699.452,E2 -20699.452} C_VEL
LIN {X 0,Y 228.93,Z 363.104,A -85,B 0,C 180,E1 -20701.76,E2 -20701.76} C_VEL
LIN {X 0,Y 225.467,Z 369.339,A -85,B 0,C 180,E1 -20704.062,E2 -20704.062} C_VEL
LIN {X 0,Y 222.447,Z 374.281,A -85,B 0,C 180,E1 -20706.349,E2 -20706.349} C_VEL
LIN {X 0,Y 219.25,Z 379.096,A -85,B 0,C 180,E1 -20709.223,E2 -20709.223} C_VEL
LIN {X 0,Y 216.186,Z 383.21,A -85,B 0,C 180,E1 -20712.762,E2 -20712.762} C_VEL
LIN {X 0,Y 214.592,Z 385.072,A -85,B 0,C 180,E1 -20715.19,E2 -20715.19} C_VEL
LIN {X 0,Y 213.484,Z 386.097,A -85,B 0,C 180,E1 -20717.308,E2 -20717.308} C_VEL
LIN {X 0,Y 212.659,Z 386.622,A -85,B 0,C 180,E1 -20719.299,E2 -20719.299} C_VEL
LIN {X 0,Y 211.867,Z 386.616,A -85,B 0,C 180,E1 -20721.747,E2 -20721.747} C_VEL
LIN {X 0,Y 211.479,Z 386.216,A -85,B 0,C 180,E1 -20723.503,E2 -20723.503} C_VEL
LIN {X 0,Y 211.134,Z 385.047,A -85,B 0,C 180,E1 -20726.003,E2 -20726.003} C_VEL
LIN {X 0,Y 211.076,Z 382.827,A -85,B 0,C 180,E1 -20728.869,E2 -20728.869} C_VEL
LIN {X 0,Y 211.347,Z 379.043,A -85,B 0,C 180,E1 -20732.145,E2 -20732.145} C_VEL
LIN {X 0,Y 211.772,Z 374.698,A -85,B 0,C 180,E1 -20734.923,E2 -20734.923} C_VEL
LIN {X 0,Y 212.437,Z 368.337,A -85,B 0,C 180,E1 -20738.067,E2 -20738.067} C_VEL
LIN {X 0,Y 213.264,Z 361.554,A -85,B 0,C 180,E1 -20740.714,E2 -20740.714} C_VEL
LIN {X 0,Y 214.485,Z 352.689,A -85,B 0,C 180,E1 -20743.481,E2 -20743.481} C_VEL
LIN {X 0,Y 215.728,Z 343.584,A -85,B 0,C 180,E1 -20745.785,E2 -20745.785} C_VEL
LIN {X 0,Y 217.093,Z 334,A -85,B 0,C 180,E1 -20747.767,E2 -20747.767} C_VEL
LIN {X 0,Y 218.734,Z 321.76,A -85,B 0,C 180,E1 -20749.779,E2 -20749.779} C_VEL
LIN {X 0,Y 220.266,Z 308.847,A -85,B 0,C 180,E1 -20751.419,E2 -20751.419} C_VEL
LIN {X 0,Y 221.461,Z 295.232,A -85,B 0,C 180,E1 -20752.69,E2 -20752.69} C_VEL
LIN {X 0,Y 222.413,Z 282.111,A -85,B 0,C 180,E1 -20753.543,E2 -20753.543} C_VEL
LIN {X 0,Y 225.653,Z 212.967,A -85,B 0,C 180,E1 -20756.426,E2 -20756.426} C_VEL
LIN {X 0,Y 216.732,Z 184.87,A -85,B 0,C 180,E1 -20758.472,E2 -20758.472} C_VEL
LIN {X 0,Y 213.791,Z 176.854,A -85,B 0,C 180,E1 -20759.149,E2 -20759.149} C_VEL
LIN {X 0,Y 213.789,Z 176.856,A -85,B 0,C 180,E1 -20762.596,E2 -20762.596} C_VEL
LIN {X 0,Y 213.8,Z 176.852,A -85,B 0,C 180,E1 -20766.989,E2 -20766.989} C_VEL
LIN {X 0,Y 213.884,Z 176.842,A -85,B 0,C 180,E1 -20772.797,E2 -20772.797} C_VEL
LIN {X 0,Y 213.917,Z 176.838,A -85,B 0,C 180,E1 -20776.703,E2 -20776.703} C_VEL
LIN {X 0,Y 214.138,Z 176.81,A -85,B 0,C 180,E1 -20780.553,E2 -20780.553} C_VEL
LIN {X 0,Y 214.078,Z 176.818,A -85,B 0,C 180,E1 -20784.346,E2 -20784.346} C_VEL
LIN {X 0,Y 214.408,Z 176.776,A -85,B 0,C 180,E1 -20788.12,E2 -20788.12} C_VEL
LIN {X 0,Y 214.516,Z 176.762,A -85,B 0,C 180,E1 -20789.998,E2 -20789.998} C_VEL
LIN {X 0,Y 214.408,Z 176.778,A -85,B 0,C 180,E1 -20791.877,E2 -20791.877} C_VEL
LIN {X 0,Y 214.18,Z 176.805,A -85,B 0,C 180,E1 -20797.54,E2 -20797.54} C_VEL
LIN {X 0,Y 213.984,Z 176.83,A -85,B 0,C 180,E1 -20801.363,E2 -20801.363} C_VEL
LIN {X 0,Y 213.873,Z 176.844,A -85,B 0,C 180,E1 -20805.24,E2 -20805.24} C_VEL
LIN {X 0,Y 213.791,Z 176.853,A -85,B 0,C 180,E1 -20809.19,E2 -20809.19} C_VEL
LIN {X 0,Y 213.783,Z 176.856,A -85,B 0,C 180,E1 -20813.232,E2 -20813.232} C_VEL
LIN {X 0,Y 213.784,Z 176.856,A -85,B 0,C 180,E1 -20817.425,E2 -20817.425} C_VEL
LIN {X 0,Y 213.758,Z 176.856,A -85,B 0,C 180,E1 -20821.737,E2 -20821.737} C_VEL
LIN {X 0,Y 213.74,Z 176.858,A -85,B 0,C 180,E1 -20826.287,E2 -20826.287} C_VEL
LIN {X 0,Y 213.695,Z 176.863,A -85,B 0,C 180,E1 -20831.127,E2 -20831.127} C_VEL
LIN {X 0,Y 213.698,Z 176.863,A -85,B 0,C 180,E1 -20833.678,E2 -20833.678} C_VEL
LIN {X 0,Y 213.698,Z 176.865,A -85,B 0,C 180,E1 -20836.344,E2 -20836.344} C_VEL
LIN {X 0,Y 213.7,Z 176.863,A -85,B 0,C 180,E1 -20841.328,E2 -20841.328} C_VEL
LIN {X 0,Y 213.75,Z 176.858,A -85,B 0,C 180,E1 -20846.016,E2 -20846.016} C_VEL
LIN {X 0,Y 213.743,Z 176.859,A -85,B 0,C 180,E1 -20850.448,E2 -20850.448} C_VEL
LIN {X 0,Y 213.745,Z 176.859,A -85,B 0,C 180,E1 -20854.694,E2 -20854.694} C_VEL
LIN {X 0,Y 213.769,Z 176.856,A -85,B 0,C 180,E1 -20858.798,E2 -20858.798} C_VEL
LIN {X 0,Y 213.873,Z 176.842,A -85,B 0,C 180,E1 -20862.797,E2 -20862.797} C_VEL
LIN {X 0,Y 213.906,Z 176.838,A -85,B 0,C 180,E1 -20866.703,E2 -20866.703} C_VEL
LIN {X 0,Y 214.127,Z 176.811,A -85,B 0,C 180,E1 -20870.554,E2 -20870.554} C_VEL
LIN {X 0,Y 214.068,Z 176.818,A -85,B 0,C 180,E1 -20874.347,E2 -20874.347} C_VEL
LIN {X 0,Y 214.397,Z 176.78,A -85,B 0,C 180,E1 -20878.121,E2 -20878.121} C_VEL
LIN {X 0,Y 214.506,Z 176.765,A -85,B 0,C 180,E1 -20880,E2 -20880} C_VEL
LIN {X 0,Y 214.397,Z 176.777,A -85,B 0,C 180,E1 -20881.878,E2 -20881.878} C_VEL
LIN {X 0,Y 214.17,Z 176.807,A -85,B 0,C 180,E1 -20887.542,E2 -20887.542} C_VEL
LIN {X 0,Y 213.975,Z 176.828,A -85,B 0,C 180,E1 -20891.365,E2 -20891.365} C_VEL
LIN {X 0,Y 213.864,Z 176.845,A -85,B 0,C 180,E1 -20895.242,E2 -20895.242} C_VEL
LIN {X 0,Y 213.783,Z 176.852,A -85,B 0,C 180,E1 -20899.192,E2 -20899.192} C_VEL
LIN {X 0,Y 213.757,Z 176.859,A -85,B 0,C 180,E1 -20903.237,E2 -20903.237} C_VEL
LIN {X 0,Y 213.778,Z 176.854,A -85,B 0,C 180,E1 -20907.427,E2 -20907.427} C_VEL
LIN {X 0,Y 213.753,Z 176.858,A -85,B 0,C 180,E1 -20911.74,E2 -20911.74} C_VEL
LIN {X 0,Y 213.735,Z 176.855,A -85,B 0,C 180,E1 -20916.29,E2 -20916.29} C_VEL
LIN {X 0,Y 213.692,Z 176.867,A -85,B 0,C 180,E1 -20921.13,E2 -20921.13} C_VEL
LIN {X 0,Y 213.66,Z 176.866,A -85,B 0,C 180,E1 -20925.795,E2 -20925.795} C_VEL
LIN {X 0,Y 213.698,Z 176.867,A -85,B 0,C 180,E1 -20929.149,E2 -20929.149} C_VEL
LIN {X 0,Y 213.784,Z 176.853,A -85,B 0,C 180,E1 -20933.917,E2 -20933.917} C_VEL
LIN {X 0,Y 213.645,Z 177.528,A -85,B 0,C 180,E1 -20934.781,E2 -20934.781} C_VEL
LIN {X 0,Y 213.138,Z 179.593,A -85,B 0,C 180,E1 -20935.794,E2 -20935.794} C_VEL
LIN {X 0,Y 212.248,Z 183.052,A -85,B 0,C 180,E1 -20936.963,E2 -20936.963} C_VEL
LIN {X 0,Y 211.494,Z 187.792,A -85,B 0,C 180,E1 -20937.918,E2 -20937.918} C_VEL
LIN {X 0,Y 211.296,Z 193.212,A -85,B 0,C 180,E1 -20938.688,E2 -20938.688} C_VEL
LIN {X 0,Y 212.273,Z 198.842,A -85,B 0,C 180,E1 -20939.245,E2 -20939.245} C_VEL
LIN {X 0,Y 215.015,Z 208.569,A -85,B 0,C 180,E1 -20939.961,E2 -20939.961} C_VEL
LIN {X 0,Y 218.07,Z 237.255,A -85,B 0,C 180,E1 -20941.553,E2 -20941.553} C_VEL
LIN {X 0,Y 215.298,Z 295.632,A -85,B 0,C 180,E1 -20944.115,E2 -20944.115} C_VEL
LIN {X 0,Y 214.117,Z 309.962,A -85,B 0,C 180,E1 -20945.133,E2 -20945.133} C_VEL
LIN {X 0,Y 212.751,Z 322.305,A -85,B 0,C 180,E1 -20946.39,E2 -20946.39} C_VEL
LIN {X 0,Y 211.272,Z 334.419,A -85,B 0,C 180,E1 -20948.025,E2 -20948.025} C_VEL
LIN {X 0,Y 209.693,Z 345.394,A -85,B 0,C 180,E1 -20949.904,E2 -20949.904} C_VEL
LIN {X 0,Y 208.096,Z 356.43,A -85,B 0,C 180,E1 -20952.306,E2 -20952.306} C_VEL
LIN {X 0,Y 206.834,Z 365.412,A -85,B 0,C 180,E1 -20954.734,E2 -20954.734} C_VEL
LIN {X 0,Y 205.672,Z 374.083,A -85,B 0,C 180,E1 -20957.67,E2 -20957.67} C_VEL
LIN {X 0,Y 205.015,Z 381.025,A -85,B 0,C 180,E1 -20960.63,E2 -20960.63} C_VEL
LIN {X 0,Y 204.626,Z 387.326,A -85,B 0,C 180,E1 -20964.088,E2 -20964.088} C_VEL
LIN {X 0,Y 204.514,Z 391.342,A -85,B 0,C 180,E1 -20967.047,E2 -20967.047} C_VEL
LIN {X 0,Y 204.592,Z 394.25,A -85,B 0,C 180,E1 -20970.002,E2 -20970.002} C_VEL
LIN {X 0,Y 204.54,Z 395.582,A -85,B 0,C 180,E1 -20971.971,E2 -20971.971} C_VEL
LIN {X 0,Y 204.43,Z 397.015,A -85,B 0,C 180,E1 -20975.921,E2 -20975.921} C_VEL
LIN {X 0,Y 204.67,Z 397.14,A -85,B 0,C 180,E1 -20977.896,E2 -20977.896} C_VEL
LIN {X 0,Y 205.822,Z 396.159,A -85,B 0,C 180,E1 -20981.824,E2 -20981.824} C_VEL
LIN {X 0,Y 207.755,Z 393.641,A -85,B 0,C 180,E1 -20985.703,E2 -20985.703} C_VEL
LIN {X 0,Y 210.022,Z 390.645,A -85,B 0,C 180,E1 -20988.538,E2 -20988.538} C_VEL
LIN {X 0,Y 212.834,Z 386.681,A -85,B 0,C 180,E1 -20991.3,E2 -20991.3} C_VEL
LIN {X 0,Y 215.998,Z 381.654,A -85,B 0,C 180,E1 -20994,E2 -20994} C_VEL
LIN {X 0,Y 219.644,Z 375.418,A -85,B 0,C 180,E1 -20996.615,E2 -20996.615} C_VEL
LIN {X 0,Y 223.994,Z 367.763,A -85,B 0,C 180,E1 -20999.101,E2 -20999.101} C_VEL
LIN {X 0,Y 228.826,Z 358.341,A -85,B 0,C 180,E1 -21001.476,E2 -21001.476} C_VEL
LIN {X 0,Y 233.666,Z 347.73,A -85,B 0,C 180,E1 -21003.552,E2 -21003.552} C_VEL
LIN {X 0,Y 237.874,Z 336.979,A -85,B 0,C 180,E1 -21005.18,E2 -21005.18} C_VEL
LIN {X 0,Y 241.854,Z 325.246,A -85,B 0,C 180,E1 -21006.565,E2 -21006.565} C_VEL
LIN {X 0,Y 245.354,Z 313.12,A -85,B 0,C 180,E1 -21007.626,E2 -21007.626} C_VEL
LIN {X 0,Y 248.516,Z 298.482,A -85,B 0,C 180,E1 -21008.555,E2 -21008.555} C_VEL
LIN {X 0,Y 250.623,Z 283.407,A -85,B 0,C 180,E1 -21009.207,E2 -21009.207} C_VEL
LIN {X 0,Y 254.335,Z 250.421,A -85,B 0,C 180,E1 -21010.469,E2 -21010.469} C_VEL
LIN {X 0,Y 251.59,Z 242.791,A -85,B 0,C 180,E1 -21012.27,E2 -21012.27} C_VEL
LIN {X 0,Y 248.649,Z 235.874,A -85,B 0,C 180,E1 -21014.334,E2 -21014.334} C_VEL
LIN {X 0,Y 246.108,Z 230.717,A -85,B 0,C 180,E1 -21016.336,E2 -21016.336} C_VEL
LIN {X 0,Y 244.086,Z 226.646,A -85,B 0,C 180,E1 -21018.246,E2 -21018.246} C_VEL
LIN {X 0,Y 241.479,Z 221.698,A -85,B 0,C 180,E1 -21021.344,E2 -21021.344} C_VEL
LIN {X 0,Y 239.305,Z 217.892,A -85,B 0,C 180,E1 -21025.492,E2 -21025.492} C_VEL
LIN {X 0,Y 238.73,Z 216.641,A -85,B 0,C 180,E1 -21028.622,E2 -21028.622} C_VEL
LIN {X 0,Y 238.98,Z 216.702,A -85,B 0,C 180,E1 -21031.453,E2 -21031.453} C_VEL
LIN {X 0,Y 240.64,Z 218.783,A -85,B 0,C 180,E1 -21035.643,E2 -21035.643} C_VEL
LIN {X 0,Y 241.764,Z 219.951,A -85,B 0,C 180,E1 -21037.158,E2 -21037.158} C_VEL
LIN {X 0,Y 244.713,Z 224.484,A -85,B 0,C 180,E1 -21040.454,E2 -21040.454} C_VEL
LIN {X 0,Y 247.492,Z 229.12,A -85,B 0,C 180,E1 -21042.839,E2 -21042.839} C_VEL
LIN {X 0,Y 250.001,Z 233.608,A -85,B 0,C 180,E1 -21044.69,E2 -21044.69} C_VEL
LIN {X 0,Y 252.847,Z 239.375,A -85,B 0,C 180,E1 -21046.525,E2 -21046.525} C_VEL
LIN {X 0,Y 254.852,Z 244.48,A -85,B 0,C 180,E1 -21047.806,E2 -21047.806} C_VEL
LIN {X 0,Y 249.739,Z 287.53,A -85,B 0,C 180,E1 -21049.463,E2 -21049.463} C_VEL
LIN {X 0,Y 247.432,Z 300.069,A -85,B 0,C 180,E1 -21050.188,E2 -21050.188} C_VEL
LIN {X 0,Y 244.68,Z 311.606,A -85,B 0,C 180,E1 -21051.119,E2 -21051.119} C_VEL
LIN {X 0,Y 241.059,Z 323.707,A -85,B 0,C 180,E1 -21052.427,E2 -21052.427} C_VEL
LIN {X 0,Y 236.967,Z 335.215,A -85,B 0,C 180,E1 -21054.042,E2 -21054.042} C_VEL
LIN {X 0,Y 232.507,Z 345.844,A -85,B 0,C 180,E1 -21055.959,E2 -21055.959} C_VEL
LIN {X 0,Y 227.739,Z 355.66,A -85,B 0,C 180,E1 -21058.232,E2 -21058.232} C_VEL
LIN {X 0,Y 223.624,Z 363.163,A -85,B 0,C 180,E1 -21060.451,E2 -21060.451} C_VEL
LIN {X 0,Y 219.271,Z 370.411,A -85,B 0,C 180,E1 -21063.216,E2 -21063.216} C_VEL
LIN {X 0,Y 214.864,Z 376.996,A -85,B 0,C 180,E1 -21066.574,E2 -21066.574} C_VEL
LIN {X 0,Y 211.671,Z 381.184,A -85,B 0,C 180,E1 -21069.557,E2 -21069.557} C_VEL
LIN {X 0,Y 208.993,Z 384.287,A -85,B 0,C 180,E1 -21072.778,E2 -21072.778} C_VEL
LIN {X 0,Y 207.12,Z 386.069,A -85,B 0,C 180,E1 -21075.752,E2 -21075.752} C_VEL
LIN {X 0,Y 206.102,Z 386.723,A -85,B 0,C 180,E1 -21077.873,E2 -21077.873} C_VEL
LIN {X 0,Y 205.268,Z 386.936,A -85,B 0,C 180,E1 -21080.023,E2 -21080.023} C_VEL
LIN {X 0,Y 204.653,Z 386.634,A -85,B 0,C 180,E1 -21082.195,E2 -21082.195} C_VEL
LIN {X 0,Y 204.212,Z 385.837,A -85,B 0,C 180,E1 -21084.393,E2 -21084.393} C_VEL
LIN {X 0,Y 203.994,Z 384.545,A -85,B 0,C 180,E1 -21086.608,E2 -21086.608} C_VEL
LIN {X 0,Y 203.978,Z 382.653,A -85,B 0,C 180,E1 -21088.841,E2 -21088.841} C_VEL
LIN {X 0,Y 204.277,Z 378.723,A -85,B 0,C 180,E1 -21092.227,E2 -21092.227} C_VEL
LIN {X 0,Y 204.795,Z 373.156,A -85,B 0,C 180,E1 -21095.69,E2 -21095.69} C_VEL
LIN {X 0,Y 205.488,Z 367.018,A -85,B 0,C 180,E1 -21098.621,E2 -21098.621} C_VEL
LIN {X 0,Y 206.448,Z 359.486,A -85,B 0,C 180,E1 -21101.499,E2 -21101.499} C_VEL
LIN {X 0,Y 207.812,Z 350.043,A -85,B 0,C 180,E1 -21104.381,E2 -21104.381} C_VEL
LIN {X 0,Y 209.275,Z 339.551,A -85,B 0,C 180,E1 -21106.923,E2 -21106.923} C_VEL
LIN {X 0,Y 210.879,Z 328.239,A -85,B 0,C 180,E1 -21109.098,E2 -21109.098} C_VEL
LIN {X 0,Y 212.483,Z 315.789,A -85,B 0,C 180,E1 -21110.963,E2 -21110.963} C_VEL
LIN {X 0,Y 213.906,Z 302.885,A -85,B 0,C 180,E1 -21112.434,E2 -21112.434} C_VEL
LIN {X 0,Y 215.02,Z 288.789,A -85,B 0,C 180,E1 -21113.593,E2 -21113.593} C_VEL
LIN {X 0,Y 215.973,Z 274.153,A -85,B 0,C 180,E1 -21114.351,E2 -21114.351} C_VEL
LIN {X 0,Y 218.837,Z 214.296,A -85,B 0,C 180,E1 -21116.908,E2 -21116.908} C_VEL
LIN {X 0,Y 210.221,Z 187.119,A -85,B 0,C 180,E1 -21118.964,E2 -21118.964} C_VEL
LIN {X 0,Y 206.735,Z 177.756,A -85,B 0,C 180,E1 -21119.763,E2 -21119.763} C_VEL
LIN {X 0,Y 206.684,Z 177.74,A -85,B 0,C 180,E1 -21123.764,E2 -21123.764} C_VEL
LIN {X 0,Y 206.718,Z 177.736,A -85,B 0,C 180,E1 -21128.037,E2 -21128.037} C_VEL
LIN {X 0,Y 206.808,Z 177.726,A -85,B 0,C 180,E1 -21132.189,E2 -21132.189} C_VEL
LIN {X 0,Y 206.858,Z 177.72,A -85,B 0,C 180,E1 -21136.24,E2 -21136.24} C_VEL
LIN {X 0,Y 207.083,Z 177.69,A -85,B 0,C 180,E1 -21140.229,E2 -21140.229} C_VEL
LIN {X 0,Y 207.042,Z 177.695,A -85,B 0,C 180,E1 -21144.154,E2 -21144.154} C_VEL
LIN {X 0,Y 207.348,Z 177.655,A -85,B 0,C 180,E1 -21148.056,E2 -21148.056} C_VEL
LIN {X 0,Y 207.484,Z 177.637,A -85,B 0,C 180,E1 -21149.998,E2 -21149.998} C_VEL
LIN {X 0,Y 207.347,Z 177.657,A -85,B 0,C 180,E1 -21151.941,E2 -21151.941} C_VEL
LIN {X 0,Y 207.124,Z 177.682,A -85,B 0,C 180,E1 -21157.799,E2 -21157.799} C_VEL
LIN {X 0,Y 206.905,Z 177.713,A -85,B 0,C 180,E1 -21161.758,E2 -21161.758} C_VEL
LIN {X 0,Y 206.805,Z 177.721,A -85,B 0,C 180,E1 -21165.774,E2 -21165.774} C_VEL
LIN {X 0,Y 206.711,Z 177.735,A -85,B 0,C 180,E1 -21169.874,E2 -21169.874} C_VEL
LIN {X 0,Y 206.7,Z 177.733,A -85,B 0,C 180,E1 -21174.078,E2 -21174.078} C_VEL
LIN {X 0,Y 206.686,Z 177.737,A -85,B 0,C 180,E1 -21178.425,E2 -21178.425} C_VEL
LIN {X 0,Y 206.693,Z 177.737,A -85,B 0,C 180,E1 -21182.956,E2 -21182.956} C_VEL
LIN {X 0,Y 206.666,Z 177.74,A -85,B 0,C 180,E1 -21187.74,E2 -21187.74} C_VEL
LIN {X 0,Y 206.628,Z 177.741,A -85,B 0,C 180,E1 -21191.557,E2 -21191.557} C_VEL
LIN {X 0,Y 206.626,Z 177.745,A -85,B 0,C 180,E1 -21195.581,E2 -21195.581} C_VEL
LIN {X 0,Y 206.643,Z 177.74,A -85,B 0,C 180,E1 -21199.744,E2 -21199.744} C_VEL
LIN {X 0,Y 206.695,Z 177.74,A -85,B 0,C 180,E1 -21204.687,E2 -21204.687} C_VEL
LIN {X 0,Y 206.69,Z 177.735,A -85,B 0,C 180,E1 -21209.333,E2 -21209.333} C_VEL
LIN {X 0,Y 206.68,Z 177.739,A -85,B 0,C 180,E1 -21213.764,E2 -21213.764} C_VEL
LIN {X 0,Y 206.707,Z 177.733,A -85,B 0,C 180,E1 -21218.037,E2 -21218.037} C_VEL
LIN {X 0,Y 206.797,Z 177.727,A -85,B 0,C 180,E1 -21222.189,E2 -21222.189} C_VEL
LIN {X 0,Y 206.847,Z 177.717,A -85,B 0,C 180,E1 -21226.241,E2 -21226.241} C_VEL
LIN {X 0,Y 207.072,Z 177.692,A -85,B 0,C 180,E1 -21230.229,E2 -21230.229} C_VEL
LIN {X 0,Y 207.032,Z 177.694,A -85,B 0,C 180,E1 -21234.154,E2 -21234.154} C_VEL
LIN {X 0,Y 207.337,Z 177.66,A -85,B 0,C 180,E1 -21238.057,E2 -21238.057} C_VEL
LIN {X 0,Y 207.474,Z 177.641,A -85,B 0,C 180,E1 -21240,E2 -21240} C_VEL
LIN {X 0,Y 207.337,Z 177.656,A -85,B 0,C 180,E1 -21241.942,E2 -21241.942} C_VEL
LIN {X 0,Y 207.115,Z 177.687,A -85,B 0,C 180,E1 -21247.801,E2 -21247.801} C_VEL
LIN {X 0,Y 206.896,Z 177.712,A -85,B 0,C 180,E1 -21251.76,E2 -21251.76} C_VEL
LIN {X 0,Y 206.797,Z 177.726,A -85,B 0,C 180,E1 -21255.776,E2 -21255.776} C_VEL
LIN {X 0,Y 206.704,Z 177.735,A -85,B 0,C 180,E1 -21259.877,E2 -21259.877} C_VEL
LIN {X 0,Y 206.685,Z 177.738,A -85,B 0,C 180,E1 -21264.082,E2 -21264.082} C_VEL
LIN {X 0,Y 206.68,Z 177.736,A -85,B 0,C 180,E1 -21268.428,E2 -21268.428} C_VEL
LIN {X 0,Y 206.688,Z 177.739,A -85,B 0,C 180,E1 -21272.959,E2 -21272.959} C_VEL
LIN {X 0,Y 206.662,Z 177.74,A -85,B 0,C 180,E1 -21277.743,E2 -21277.743} C_VEL
LIN {X 0,Y 206.625,Z 177.745,A -85,B 0,C 180,E1 -21281.56,E2 -21281.56} C_VEL
LIN {X 0,Y 206.624,Z 177.747,A -85,B 0,C 180,E1 -21285.584,E2 -21285.584} C_VEL
LIN {X 0,Y 206.642,Z 177.744,A -85,B 0,C 180,E1 -21289.747,E2 -21289.747} C_VEL
LIN {X 0,Y 206.77,Z 177.76,A -85,B 0,C 180,E1 -21294.354,E2 -21294.354} C_VEL
LIN {X 0,Y 208.462,Z 186.443,A -85,B 0,C 180,E1 -21298.269,E2 -21298.269} C_VEL
LIN {X 0,Y 212.273,Z 198.842,A -85,B 0,C 180,E1 -21299.245,E2 -21299.245} C_VEL
LIN {X 0,Y 213.015,Z 202.59,A -85,B 0,C 180,E1 -21299.495,E2 -21299.495} C_VEL
LIN {X 0,Y 213.08,Z 206.47,A -85,B 0,C 180,E1 -21299.688,E2 -21299.688} C_VEL
LIN {X 0,Y 211.996,Z 214.325,A -85,B 0,C 180,E1 -21299.971,E2 -21299.971} C_VEL
LIN {X 0,Y 210.346,Z 224.215,A -85,B 0,C 180,E1 -21300.307,E2 -21300.307} C_VEL
LIN {X 0,Y 210.437,Z 230.121,A -85,B 0,C 180,E1 -21300.601,E2 -21300.601} C_VEL
LIN {X 0,Y 211.266,Z 237.779,A -85,B 0,C 180,E1 -21301.038,E2 -21301.038} C_VEL
LIN {X 0,Y 208.405,Z 295.52,A -85,B 0,C 180,E1 -21303.664,E2 -21303.664} C_VEL
LIN {X 0,Y 207.26,Z 309.05,A -85,B 0,C 180,E1 -21304.655,E2 -21304.655} C_VEL
LIN {X 0,Y 206.008,Z 320.596,A -85,B 0,C 180,E1 -21305.836,E2 -21305.836} C_VEL
LIN {X 0,Y 204.461,Z 332.963,A -85,B 0,C 180,E1 -21307.519,E2 -21307.519} C_VEL
LIN {X 0,Y 202.818,Z 344.032,A -85,B 0,C 180,E1 -21309.439,E2 -21309.439} C_VEL
LIN {X 0,Y 201.286,Z 354.368,A -85,B 0,C 180,E1 -21311.687,E2 -21311.687} C_VEL
LIN {X 0,Y 199.965,Z 363.627,A -85,B 0,C 180,E1 -21314.196,E2 -21314.196} C_VEL
LIN {X 0,Y 198.718,Z 372.651,A -85,B 0,C 180,E1 -21317.232,E2 -21317.232} C_VEL
LIN {X 0,Y 197.986,Z 379.837,A -85,B 0,C 180,E1 -21320.295,E2 -21320.295} C_VEL
LIN {X 0,Y 197.567,Z 386.359,A -85,B 0,C 180,E1 -21323.876,E2 -21323.876} C_VEL
LIN {X 0,Y 197.469,Z 390.568,A -85,B 0,C 180,E1 -21326.942,E2 -21326.942} C_VEL
LIN {X 0,Y 197.531,Z 393.633,A -85,B 0,C 180,E1 -21330.002,E2 -21330.002} C_VEL
LIN {X 0,Y 197.47,Z 395.098,A -85,B 0,C 180,E1 -21332.041,E2 -21332.041} C_VEL
LIN {X 0,Y 197.36,Z 396.682,A -85,B 0,C 180,E1 -21336.134,E2 -21336.134} C_VEL
LIN {X 0,Y 198.136,Z 396.732,A -85,B 0,C 180,E1 -21340.217,E2 -21340.217} C_VEL
LIN {X 0,Y 198.86,Z 396.162,A -85,B 0,C 180,E1 -21342.244,E2 -21342.244} C_VEL
LIN {X 0,Y 200.911,Z 393.832,A -85,B 0,C 180,E1 -21346.253,E2 -21346.253} C_VEL
LIN {X 0,Y 203.33,Z 391.042,A -85,B 0,C 180,E1 -21349.171,E2 -21349.171} C_VEL
LIN {X 0,Y 206.267,Z 387.275,A -85,B 0,C 180,E1 -21352.013,E2 -21352.013} C_VEL
LIN {X 0,Y 209.591,Z 382.451,A -85,B 0,C 180,E1 -21354.783,E2 -21354.783} C_VEL
LIN {X 0,Y 213.411,Z 376.519,A -85,B 0,C 180,E1 -21357.456,E2 -21357.456} C_VEL
LIN {X 0,Y 217.94,Z 369.182,A -85,B 0,C 180,E1 -21359.991,E2 -21359.991} C_VEL
LIN {X 0,Y 222.967,Z 360.185,A -85,B 0,C 180,E1 -21362.403,E2 -21362.403} C_VEL
LIN {X 0,Y 228.431,Z 349.019,A -85,B 0,C 180,E1 -21364.695,E2 -21364.695} C_VEL
LIN {X 0,Y 233.323,Z 337.512,A -85,B 0,C 180,E1 -21366.507,E2 -21366.507} C_VEL
LIN {X 0,Y 237.481,Z 325.969,A -85,B 0,C 180,E1 -21367.886,E2 -21367.886} C_VEL
LIN {X 0,Y 241.385,Z 313.068,A -85,B 0,C 180,E1 -21369.024,E2 -21369.024} C_VEL
LIN {X 0,Y 244.685,Z 298.402,A -85,B 0,C 180,E1 -21369.949,E2 -21369.949} C_VEL
LIN {X 0,Y 246.956,Z 283.1,A -85,B 0,C 180,E1 -21370.612,E2 -21370.612} C_VEL
LIN {X 0,Y 250.505,Z 253.438,A -85,B 0,C 180,E1 -21371.769,E2 -21371.769} C_VEL
LIN {X 0,Y 247.473,Z 245.135,A -85,B 0,C 180,E1 -21373.958,E2 -21373.958} C_VEL
LIN {X 0,Y 245.392,Z 240.231,A -85,B 0,C 180,E1 -21375.633,E2 -21375.633} C_VEL
LIN {X 0,Y 243.789,Z 236.741,A -85,B 0,C 180,E1 -21377.038,E2 -21377.038} C_VEL
LIN {X 0,Y 242.112,Z 233.119,A -85,B 0,C 180,E1 -21378.763,E2 -21378.763} C_VEL
LIN {X 0,Y 239.725,Z 228.322,A -85,B 0,C 180,E1 -21381.84,E2 -21381.84} C_VEL
LIN {X 0,Y 237.888,Z 224.828,A -85,B 0,C 180,E1 -21385.66,E2 -21385.66} C_VEL
LIN {X 0,Y 237.414,Z 223.631,A -85,B 0,C 180,E1 -21388.428,E2 -21388.428} C_VEL
LIN {X 0,Y 237.695,Z 223.788,A -85,B 0,C 180,E1 -21391.766,E2 -21391.766} C_VEL
LIN {X 0,Y 239.473,Z 225.97,A -85,B 0,C 180,E1 -21395.917,E2 -21395.917} C_VEL
LIN {X 0,Y 240.188,Z 226.902,A -85,B 0,C 180,E1 -21396.924,E2 -21396.924} C_VEL
LIN {X 0,Y 242.73,Z 230.956,A -85,B 0,C 180,E1 -21399.941,E2 -21399.941} C_VEL
LIN {X 0,Y 245.268,Z 235.479,A -85,B 0,C 180,E1 -21402.3,E2 -21402.3} C_VEL
LIN {X 0,Y 247.552,Z 239.709,A -85,B 0,C 180,E1 -21404.06,E2 -21404.06} C_VEL
LIN {X 0,Y 249.924,Z 244.848,A -85,B 0,C 180,E1 -21405.742,E2 -21405.742} C_VEL
LIN {X 0,Y 251.036,Z 247.966,A -85,B 0,C 180,E1 -21406.523,E2 -21406.523} C_VEL
LIN {X 0,Y 246.03,Z 287.408,A -85,B 0,C 180,E1 -21408.052,E2 -21408.052} C_VEL
LIN {X 0,Y 243.617,Z 299.977,A -85,B 0,C 180,E1 -21408.776,E2 -21408.776} C_VEL
LIN {X 0,Y 240.744,Z 311.634,A -85,B 0,C 180,E1 -21409.706,E2 -21409.706} C_VEL
LIN {X 0,Y 236.874,Z 324.053,A -85,B 0,C 180,E1 -21411.039,E2 -21411.039} C_VEL
LIN {X 0,Y 232.472,Z 335.744,A -85,B 0,C 180,E1 -21412.688,E2 -21412.688} C_VEL
LIN {X 0,Y 228.115,Z 345.549,A -85,B 0,C 180,E1 -21414.475,E2 -21414.475} C_VEL
LIN {X 0,Y 222.858,Z 355.768,A -85,B 0,C 180,E1 -21416.837,E2 -21416.837} C_VEL
LIN {X 0,Y 217.884,Z 364.29,A -85,B 0,C 180,E1 -21419.414,E2 -21419.414} C_VEL
LIN {X 0,Y 213.794,Z 370.582,A -85,B 0,C 180,E1 -21421.884,E2 -21421.884} C_VEL
LIN {X 0,Y 209.66,Z 376.301,A -85,B 0,C 180,E1 -21424.808,E2 -21424.808} C_VEL
LIN {X 0,Y 205.866,Z 381.05,A -85,B 0,C 180,E1 -21428.09,E2 -21428.09} C_VEL
LIN {X 0,Y 204.098,Z 383.016,A -85,B 0,C 180,E1 -21429.915,E2 -21429.915} C_VEL
LIN {X 0,Y 201.788,Z 385.27,A -85,B 0,C 180,E1 -21432.78,E2 -21432.78} C_VEL
LIN {X 0,Y 199.654,Z 386.825,A -85,B 0,C 180,E1 -21436.357,E2 -21436.357} C_VEL
LIN {X 0,Y 198.664,Z 387.138,A -85,B 0,C 180,E1 -21438.566,E2 -21438.566} C_VEL
LIN {X 0,Y 197.524,Z 386.619,A -85,B 0,C 180,E1 -21442.314,E2 -21442.314} C_VEL
LIN {X 0,Y 197.003,Z 385.193,A -85,B 0,C 180,E1 -21445.347,E2 -21445.347} C_VEL
LIN {X 0,Y 196.883,Z 382.464,A -85,B 0,C 180,E1 -21448.81,E2 -21448.81} C_VEL
LIN {X 0,Y 197.206,Z 378.39,A -85,B 0,C 180,E1 -21452.315,E2 -21452.315} C_VEL
LIN {X 0,Y 197.783,Z 372.348,A -85,B 0,C 180,E1 -21456.033,E2 -21456.033} C_VEL
LIN {X 0,Y 198.427,Z 366.562,A -85,B 0,C 180,E1 -21458.81,E2 -21458.81} C_VEL
LIN {X 0,Y 199.541,Z 358.259,A -85,B 0,C 180,E1 -21462.006,E2 -21462.006} C_VEL
LIN {X 0,Y 200.851,Z 349.171,A -85,B 0,C 180,E1 -21464.775,E2 -21464.775} C_VEL
LIN {X 0,Y 202.278,Z 339.258,A -85,B 0,C 180,E1 -21467.222,E2 -21467.222} C_VEL
LIN {X 0,Y 203.832,Z 328.585,A -85,B 0,C 180,E1 -21469.337,E2 -21469.337} C_VEL
LIN {X 0,Y 205.501,Z 316.118,A -85,B 0,C 180,E1 -21471.277,E2 -21471.277} C_VEL
LIN {X 0,Y 206.84,Z 304.291,A -85,B 0,C 180,E1 -21472.702,E2 -21472.702} C_VEL
LIN {X 0,Y 207.995,Z 290.372,A -85,B 0,C 180,E1 -21473.925,E2 -21473.925} C_VEL
LIN {X 0,Y 208.915,Z 276.717,A -85,B 0,C 180,E1 -21474.715,E2 -21474.715} C_VEL
LIN {X 0,Y 212.066,Z 215.725,A -85,B 0,C 180,E1 -21477.414,E2 -21477.414} C_VEL
LIN {X 0,Y 203.797,Z 189.608,A -85,B 0,C 180,E1 -21479.445,E2 -21479.445} C_VEL
LIN {X 0,Y 199.703,Z 178.794,A -85,B 0,C 180,E1 -21480.408,E2 -21480.408} C_VEL
LIN {X 0,Y 199.627,Z 178.618,A -85,B 0,C 180,E1 -21485.008,E2 -21485.008} C_VEL
LIN {X 0,Y 199.649,Z 178.614,A -85,B 0,C 180,E1 -21489.387,E2 -21489.387} C_VEL
LIN {X 0,Y 199.748,Z 178.604,A -85,B 0,C 180,E1 -21493.65,E2 -21493.65} C_VEL
LIN {X 0,Y 200.027,Z 178.571,A -85,B 0,C 180,E1 -21499.88,E2 -21499.88} C_VEL
LIN {X 0,Y 200.006,Z 178.572,A -85,B 0,C 180,E1 -21503.947,E2 -21503.947} C_VEL
LIN {X 0,Y 200.29,Z 178.535,A -85,B 0,C 180,E1 -21507.987,E2 -21507.987} C_VEL
LIN {X 0,Y 200.451,Z 178.513,A -85,B 0,C 180,E1 -21509.998,E2 -21509.998} C_VEL
LIN {X 0,Y 199.992,Z 178.573,A -85,B 0,C 180,E1 -21514.028,E2 -21514.028} C_VEL
LIN {X 0,Y 200.072,Z 178.559,A -85,B 0,C 180,E1 -21518.076,E2 -21518.076} C_VEL
LIN {X 0,Y 199.855,Z 178.589,A -85,B 0,C 180,E1 -21522.179,E2 -21522.179} C_VEL
LIN {X 0,Y 199.744,Z 178.599,A -85,B 0,C 180,E1 -21526.347,E2 -21526.347} C_VEL
LIN {X 0,Y 199.642,Z 178.615,A -85,B 0,C 180,E1 -21530.61,E2 -21530.61} C_VEL
LIN {X 0,Y 199.625,Z 178.616,A -85,B 0,C 180,E1 -21534.989,E2 -21534.989} C_VEL
LIN {X 0,Y 199.607,Z 178.621,A -85,B 0,C 180,E1 -21539.531,E2 -21539.531} C_VEL
LIN {X 0,Y 199.664,Z 178.611,A -85,B 0,C 180,E1 -21542.35,E2 -21542.35} C_VEL
LIN {X 0,Y 199.615,Z 178.62,A -85,B 0,C 180,E1 -21546.762,E2 -21546.762} C_VEL
LIN {X 0,Y 199.592,Z 178.622,A -85,B 0,C 180,E1 -21549.33,E2 -21549.33} C_VEL
LIN {X 0,Y 199.563,Z 178.621,A -85,B 0,C 180,E1 -21552.305,E2 -21552.305} C_VEL
LIN {X 0,Y 199.573,Z 178.625,A -85,B 0,C 180,E1 -21555.226,E2 -21555.226} C_VEL
LIN {X 0,Y 199.566,Z 178.624,A -85,B 0,C 180,E1 -21558.001,E2 -21558.001} C_VEL
LIN {X 0,Y 199.593,Z 178.62,A -85,B 0,C 180,E1 -21560.771,E2 -21560.771} C_VEL
LIN {X 0,Y 199.606,Z 178.619,A -85,B 0,C 180,E1 -21565.711,E2 -21565.711} C_VEL
LIN {X 0,Y 199.681,Z 178.609,A -85,B 0,C 180,E1 -21568.133,E2 -21568.133} C_VEL
LIN {X 0,Y 199.63,Z 178.619,A -85,B 0,C 180,E1 -21572.763,E2 -21572.763} C_VEL
LIN {X 0,Y 199.665,Z 178.609,A -85,B 0,C 180,E1 -21577.22,E2 -21577.22} C_VEL
LIN {X 0,Y 199.74,Z 178.604,A -85,B 0,C 180,E1 -21581.802,E2 -21581.802} C_VEL
LIN {X 0,Y 199.765,Z 178.597,A -85,B 0,C 180,E1 -21585.743,E2 -21585.743} C_VEL
LIN {X 0,Y 200.017,Z 178.57,A -85,B 0,C 180,E1 -21589.881,E2 -21589.881} C_VEL
LIN {X 0,Y 199.995,Z 178.57,A -85,B 0,C 180,E1 -21593.948,E2 -21593.948} C_VEL
LIN {X 0,Y 200.279,Z 178.539,A -85,B 0,C 180,E1 -21597.989,E2 -21597.989} C_VEL
LIN {X 0,Y 200.441,Z 178.517,A -85,B 0,C 180,E1 -21600,E2 -21600} C_VEL
LIN {X 0,Y 199.982,Z 178.575,A -85,B 0,C 180,E1 -21604.03,E2 -21604.03} C_VEL
LIN {X 0,Y 200.063,Z 178.563,A -85,B 0,C 180,E1 -21608.077,E2 -21608.077} C_VEL
LIN {X 0,Y 199.846,Z 178.59,A -85,B 0,C 180,E1 -21612.181,E2 -21612.181} C_VEL
LIN {X 0,Y 199.736,Z 178.603,A -85,B 0,C 180,E1 -21616.349,E2 -21616.349} C_VEL
LIN {X 0,Y 199.635,Z 178.614,A -85,B 0,C 180,E1 -21620.612,E2 -21620.612} C_VEL
LIN {X 0,Y 199.614,Z 178.619,A -85,B 0,C 180,E1 -21624.992,E2 -21624.992} C_VEL
LIN {X 0,Y 199.601,Z 178.622,A -85,B 0,C 180,E1 -21629.534,E2 -21629.534} C_VEL
LIN {X 0,Y 199.659,Z 178.613,A -85,B 0,C 180,E1 -21632.353,E2 -21632.353} C_VEL
LIN {X 0,Y 199.611,Z 178.615,A -85,B 0,C 180,E1 -21636.765,E2 -21636.765} C_VEL
LIN {X 0,Y 199.589,Z 178.624,A -85,B 0,C 180,E1 -21639.332,E2 -21639.332} C_VEL
LIN {X 0,Y 199.56,Z 178.624,A -85,B 0,C 180,E1 -21642.308,E2 -21642.308} C_VEL
LIN {X 0,Y 199.57,Z 178.627,A -85,B 0,C 180,E1 -21645.229,E2 -21645.229} C_VEL
LIN {X 0,Y 199.565,Z 178.626,A -85,B 0,C 180,E1 -21648.004,E2 -21648.004} C_VEL
LIN {X 0,Y 199.664,Z 178.614,A -85,B 0,C 180,E1 -21653.248,E2 -21653.248} C_VEL
LIN {X 0,Y 199.721,Z 178.732,A -85,B 0,C 180,E1 -21654.032,E2 -21654.032} C_VEL
LIN {X 0,Y 201.232,Z 186.301,A -85,B 0,C 180,E1 -21657.572,E2 -21657.572} C_VEL
LIN {X 0,Y 208.324,Z 209.741,A -85,B 0,C 180,E1 -21659.423,E2 -21659.423} C_VEL
LIN {X 0,Y 210.437,Z 230.121,A -85,B 0,C 180,E1 -21660.601,E2 -21660.601} C_VEL
LIN {X 0,Y 210.163,Z 233.987,A -85,B 0,C 180,E1 -21660.764,E2 -21660.764} C_VEL
LIN {X 0,Y 207.608,Z 240.169,A -85,B 0,C 180,E1 -21660.861,E2 -21660.861} C_VEL
LIN {X 0,Y 204.681,Z 246.371,A -85,B 0,C 180,E1 -21660.941,E2 -21660.941} C_VEL
LIN {X 0,Y 203.871,Z 250.31,A -85,B 0,C 180,E1 -21661.076,E2 -21661.076} C_VEL
LIN {X 0,Y 201.472,Z 295.694,A -85,B 0,C 180,E1 -21663.245,E2 -21663.245} C_VEL
LIN {X 0,Y 200.307,Z 309.105,A -85,B 0,C 180,E1 -21664.268,E2 -21664.268} C_VEL
LIN {X 0,Y 199.03,Z 320.58,A -85,B 0,C 180,E1 -21665.489,E2 -21665.489} C_VEL
LIN {X 0,Y 197.443,Z 332.9,A -85,B 0,C 180,E1 -21667.228,E2 -21667.228} C_VEL
LIN {X 0,Y 195.806,Z 343.644,A -85,B 0,C 180,E1 -21669.155,E2 -21669.155} C_VEL
LIN {X 0,Y 194.212,Z 354.258,A -85,B 0,C 180,E1 -21671.542,E2 -21671.542} C_VEL
LIN {X 0,Y 192.879,Z 363.508,A -85,B 0,C 180,E1 -21674.142,E2 -21674.142} C_VEL
LIN {X 0,Y 191.596,Z 372.516,A -85,B 0,C 180,E1 -21677.288,E2 -21677.288} C_VEL
LIN {X 0,Y 190.889,Z 379.69,A -85,B 0,C 180,E1 -21680.465,E2 -21680.465} C_VEL
LIN {X 0,Y 190.503,Z 385.368,A -85,B 0,C 180,E1 -21683.648,E2 -21683.648} C_VEL
LIN {X 0,Y 190.404,Z 389.179,A -85,B 0,C 180,E1 -21686.353,E2 -21686.353} C_VEL
LIN {X 0,Y 190.442,Z 392.018,A -85,B 0,C 180,E1 -21688.945,E2 -21688.945} C_VEL
LIN {X 0,Y 190.402,Z 394.515,A -85,B 0,C 180,E1 -21692.117,E2 -21692.117} C_VEL
LIN {X 0,Y 190.214,Z 395.641,A -85,B 0,C 180,E1 -21694.24,E2 -21694.24} C_VEL
LIN {X 0,Y 190.295,Z 396.348,A -85,B 0,C 180,E1 -21696.363,E2 -21696.363} C_VEL
LIN {X 0,Y 191.128,Z 396.569,A -85,B 0,C 180,E1 -21700.596,E2 -21700.596} C_VEL
LIN {X 0,Y 192.867,Z 395.287,A -85,B 0,C 180,E1 -21704.78,E2 -21704.78} C_VEL
LIN {X 0,Y 194.092,Z 394.043,A -85,B 0,C 180,E1 -21706.84,E2 -21706.84} C_VEL
LIN {X 0,Y 196.665,Z 391.438,A -85,B 0,C 180,E1 -21709.848,E2 -21709.848} C_VEL
LIN {X 0,Y 200.844,Z 386.453,A -85,B 0,C 180,E1 -21713.731,E2 -21713.731} C_VEL
LIN {X 0,Y 205.01,Z 380.733,A -85,B 0,C 180,E1 -21716.961,E2 -21716.961} C_VEL
LIN {X 0,Y 209.5,Z 374.302,A -85,B 0,C 180,E1 -21719.659,E2 -21719.659} C_VEL
LIN {X 0,Y 215.372,Z 365.061,A -85,B 0,C 180,E1 -21722.578,E2 -21722.578} C_VEL
LIN {X 0,Y 219.943,Z 357.021,A -85,B 0,C 180,E1 -21724.555,E2 -21724.555} C_VEL
LIN {X 0,Y 224.809,Z 347.379,A -85,B 0,C 180,E1 -21726.442,E2 -21726.442} C_VEL
LIN {X 0,Y 229.942,Z 335.443,A -85,B 0,C 180,E1 -21728.239,E2 -21728.239} C_VEL
LIN {X 0,Y 234.393,Z 323.56,A -85,B 0,C 180,E1 -21729.582,E2 -21729.582} C_VEL
LIN {X 0,Y 238.202,Z 311.105,A -85,B 0,C 180,E1 -21730.614,E2 -21730.614} C_VEL
LIN {X 0,Y 241.26,Z 297.874,A -85,B 0,C 180,E1 -21731.439,E2 -21731.439} C_VEL
LIN {X 0,Y 243.569,Z 282.961,A -85,B 0,C 180,E1 -21732.075,E2 -21732.075} C_VEL
LIN {X 0,Y 246.812,Z 256.679,A -85,B 0,C 180,E1 -21733.112,E2 -21733.112} C_VEL
LIN {X 0,Y 244.511,Z 249.979,A -85,B 0,C 180,E1 -21735.016,E2 -21735.016} C_VEL
LIN {X 0,Y 242.031,Z 243.775,A -85,B 0,C 180,E1 -21737.283,E2 -21737.283} C_VEL
LIN {X 0,Y 239.991,Z 239.273,A -85,B 0,C 180,E1 -21739.472,E2 -21739.472} C_VEL
LIN {X 0,Y 237.996,Z 234.873,A -85,B 0,C 180,E1 -21742.352,E2 -21742.352} C_VEL
LIN {X 0,Y 236.414,Z 231.672,A -85,B 0,C 180,E1 -21745.999,E2 -21745.999} C_VEL
LIN {X 0,Y 236.062,Z 230.592,A -85,B 0,C 180,E1 -21748.555,E2 -21748.555} C_VEL
LIN {X 0,Y 236.322,Z 230.716,A -85,B 0,C 180,E1 -21751.587,E2 -21751.587} C_VEL
LIN {X 0,Y 237.88,Z 232.77,A -85,B 0,C 180,E1 -21755.568,E2 -21755.568} C_VEL
LIN {X 0,Y 238.711,Z 233.987,A -85,B 0,C 180,E1 -21756.823,E2 -21756.823} C_VEL
LIN {X 0,Y 240.922,Z 237.665,A -85,B 0,C 180,E1 -21759.578,E2 -21759.578} C_VEL
LIN {X 0,Y 243.244,Z 242.115,A -85,B 0,C 180,E1 -21761.884,E2 -21761.884} C_VEL
LIN {X 0,Y 245.174,Z 245.898,A -85,B 0,C 180,E1 -21763.456,E2 -21763.456} C_VEL
LIN {X 0,Y 247.332,Z 251.017,A -85,B 0,C 180,E1 -21765.145,E2 -21765.145} C_VEL
LIN {X 0,Y 242.535,Z 287.789,A -85,B 0,C 180,E1 -21766.596,E2 -21766.596} C_VEL
LIN {X 0,Y 239.733,Z 301.682,A -85,B 0,C 180,E1 -21767.415,E2 -21767.415} C_VEL
LIN {X 0,Y 236.436,Z 313.766,A -85,B 0,C 180,E1 -21768.425,E2 -21768.425} C_VEL
LIN {X 0,Y 232.371,Z 325.764,A -85,B 0,C 180,E1 -21769.765,E2 -21769.765} C_VEL
LIN {X 0,Y 227.728,Z 337.215,A -85,B 0,C 180,E1 -21771.431,E2 -21771.431} C_VEL
LIN {X 0,Y 223.174,Z 346.81,A -85,B 0,C 180,E1 -21773.218,E2 -21773.218} C_VEL
LIN {X 0,Y 217.753,Z 356.672,A -85,B 0,C 180,E1 -21775.559,E2 -21775.559} C_VEL
LIN {X 0,Y 212.652,Z 364.788,A -85,B 0,C 180,E1 -21778.106,E2 -21778.106} C_VEL
LIN {X 0,Y 208.414,Z 370.819,A -85,B 0,C 180,E1 -21780.483,E2 -21780.483} C_VEL
LIN {X 0,Y 204.171,Z 376.384,A -85,B 0,C 180,E1 -21783.372,E2 -21783.372} C_VEL
LIN {X 0,Y 199.706,Z 381.465,A -85,B 0,C 180,E1 -21786.987,E2 -21786.987} C_VEL
LIN {X 0,Y 196.5,Z 384.586,A -85,B 0,C 180,E1 -21790.302,E2 -21790.302} C_VEL
LIN {X 0,Y 194.591,Z 386.106,A -85,B 0,C 180,E1 -21792.793,E2 -21792.793} C_VEL
LIN {X 0,Y 193.372,Z 386.885,A -85,B 0,C 180,E1 -21794.739,E2 -21794.739} C_VEL
LIN {X 0,Y 191.88,Z 387.371,A -85,B 0,C 180,E1 -21797.762,E2 -21797.762} C_VEL
LIN {X 0,Y 190.564,Z 386.818,A -85,B 0,C 180,E1 -21801.642,E2 -21801.642} C_VEL
LIN {X 0,Y 190.057,Z 385.813,A -85,B 0,C 180,E1 -21804.002,E2 -21804.002} C_VEL
LIN {X 0,Y 189.795,Z 383.574,A -85,B 0,C 180,E1 -21807.285,E2 -21807.285} C_VEL
LIN {X 0,Y 189.978,Z 379.524,A -85,B 0,C 180,E1 -21811.193,E2 -21811.193} C_VEL
LIN {X 0,Y 190.464,Z 374.463,A -85,B 0,C 180,E1 -21814.716,E2 -21814.716} C_VEL
LIN {X 0,Y 191.144,Z 368.291,A -85,B 0,C 180,E1 -21818.016,E2 -21818.016} C_VEL
LIN {X 0,Y 192.078,Z 360.713,A -85,B 0,C 180,E1 -21821.195,E2 -21821.195} C_VEL
LIN {X 0,Y 193.493,Z 351.23,A -85,B 0,C 180,E1 -21824.363,E2 -21824.363} C_VEL
LIN {X 0,Y 194.976,Z 341.016,A -85,B 0,C 180,E1 -21827.06,E2 -21827.06} C_VEL
LIN {X 0,Y 196.67,Z 329.733,A -85,B 0,C 180,E1 -21829.441,E2 -21829.441} C_VEL
LIN {X 0,Y 198.336,Z 317.676,A -85,B 0,C 180,E1 -21831.425,E2 -21831.425} C_VEL
LIN {X 0,Y 199.911,Z 304.316,A -85,B 0,C 180,E1 -21833.112,E2 -21833.112} C_VEL
LIN {X 0,Y 201.111,Z 290.072,A -85,B 0,C 180,E1 -21834.395,E2 -21834.395} C_VEL
LIN {X 0,Y 202.064,Z 276.298,A -85,B 0,C 180,E1 -21835.202,E2 -21835.202} C_VEL
LIN {X 0,Y 205.213,Z 216.936,A -85,B 0,C 180,E1 -21837.932,E2 -21837.932} C_VEL
LIN {X 0,Y 197.529,Z 192.563,A -85,B 0,C 180,E1 -21839.902,E2 -21839.902} C_VEL
LIN {X 0,Y 192.625,Z 179.491,A -85,B 0,C 180,E1 -21841.123,E2 -21841.123} C_VEL
LIN {X 0,Y 192.661,Z 179.487,A -85,B 0,C 180,E1 -21846.341,E2 -21846.341} C_VEL
LIN {X 0,Y 192.699,Z 179.481,A -85,B 0,C 180,E1 -21851.49,E2 -21851.49} C_VEL
LIN {X 0,Y 192.779,Z 179.471,A -85,B 0,C 180,E1 -21857.363,E2 -21857.363} C_VEL
LIN {X 0,Y 193.03,Z 179.44,A -85,B 0,C 180,E1 -21861.624,E2 -21861.624} C_VEL
LIN {X 0,Y 193.234,Z 179.414,A -85,B 0,C 180,E1 -21867.914,E2 -21867.914} C_VEL
LIN {X 0,Y 193.417,Z 179.389,A -85,B 0,C 180,E1 -21869.998,E2 -21869.998} C_VEL
LIN {X 0,Y 192.939,Z 179.451,A -85,B 0,C 180,E1 -21874.176,E2 -21874.176} C_VEL
LIN {X 0,Y 193.024,Z 179.436,A -85,B 0,C 180,E1 -21878.372,E2 -21878.372} C_VEL
LIN {X 0,Y 192.777,Z 179.47,A -85,B 0,C 180,E1 -21882.633,E2 -21882.633} C_VEL
LIN {X 0,Y 192.695,Z 179.479,A -85,B 0,C 180,E1 -21888.506,E2 -21888.506} C_VEL
LIN {X 0,Y 192.619,Z 179.487,A -85,B 0,C 180,E1 -21894.192,E2 -21894.192} C_VEL
LIN {X 0,Y 192.6,Z 179.494,A -85,B 0,C 180,E1 -21898.863,E2 -21898.863} C_VEL
LIN {X 0,Y 192.593,Z 179.492,A -85,B 0,C 180,E1 -21903.185,E2 -21903.185} C_VEL
LIN {X 0,Y 192.539,Z 179.5,A -85,B 0,C 180,E1 -21908.352,E2 -21908.352} C_VEL
LIN {X 0,Y 192.482,Z 179.507,A -85,B 0,C 180,E1 -21913.092,E2 -21913.092} C_VEL
LIN {X 0,Y 192.481,Z 179.509,A -85,B 0,C 180,E1 -21916.905,E2 -21916.905} C_VEL
LIN {X 0,Y 192.538,Z 179.498,A -85,B 0,C 180,E1 -21921.644,E2 -21921.644} C_VEL
LIN {X 0,Y 192.59,Z 179.493,A -85,B 0,C 180,E1 -21926.812,E2 -21926.812} C_VEL
LIN {X 0,Y 192.614,Z 179.49,A -85,B 0,C 180,E1 -21931.683,E2 -21931.683} C_VEL
LIN {X 0,Y 192.657,Z 179.484,A -85,B 0,C 180,E1 -21936.342,E2 -21936.342} C_VEL
LIN {X 0,Y 192.689,Z 179.481,A -85,B 0,C 180,E1 -21941.491,E2 -21941.491} C_VEL
LIN {X 0,Y 192.769,Z 179.47,A -85,B 0,C 180,E1 -21947.364,E2 -21947.364} C_VEL
LIN {X 0,Y 193.019,Z 179.441,A -85,B 0,C 180,E1 -21951.625,E2 -21951.625} C_VEL
LIN {X 0,Y 193.223,Z 179.418,A -85,B 0,C 180,E1 -21957.915,E2 -21957.915} C_VEL
LIN {X 0,Y 193.407,Z 179.393,A -85,B 0,C 180,E1 -21960,E2 -21960} C_VEL
LIN {X 0,Y 192.929,Z 179.452,A -85,B 0,C 180,E1 -21964.178,E2 -21964.178} C_VEL
LIN {X 0,Y 193.015,Z 179.44,A -85,B 0,C 180,E1 -21968.374,E2 -21968.374} C_VEL
LIN {X 0,Y 192.768,Z 179.47,A -85,B 0,C 180,E1 -21972.635,E2 -21972.635} C_VEL
LIN {X 0,Y 192.688,Z 179.478,A -85,B 0,C 180,E1 -21978.509,E2 -21978.509} C_VEL
LIN {X 0,Y 192.604,Z 179.492,A -85,B 0,C 180,E1 -21984.189,E2 -21984.189} C_VEL
LIN {X 0,Y 192.594,Z 179.491,A -85,B 0,C 180,E1 -21988.866,E2 -21988.866} C_VEL
LIN {X 0,Y 192.588,Z 179.496,A -85,B 0,C 180,E1 -21993.187,E2 -21993.187} C_VEL
LIN {X 0,Y 192.536,Z 179.499,A -85,B 0,C 180,E1 -21998.355,E2 -21998.355} C_VEL
LIN {X 0,Y 192.479,Z 179.509,A -85,B 0,C 180,E1 -22003.095,E2 -22003.095} C_VEL
LIN {X 0,Y 192.479,Z 179.51,A -85,B 0,C 180,E1 -22006.908,E2 -22006.908} C_VEL
LIN {X 0,Y 192.552,Z 179.499,A -85,B 0,C 180,E1 -22011.651,E2 -22011.651} C_VEL
LIN {X 0,Y 192.659,Z 179.563,A -85,B 0,C 180,E1 -22013.631,E2 -22013.631} C_VEL
LIN {X 0,Y 194.001,Z 186.22,A -85,B 0,C 180,E1 -22016.839,E2 -22016.839} C_VEL
LIN {X 0,Y 201.671,Z 211.478,A -85,B 0,C 180,E1 -22018.92,E2 -22018.92} C_VEL
LIN {X 0,Y 204.434,Z 238.516,A -85,B 0,C 180,E1 -22020.53,E2 -22020.53} C_VEL
LIN {X 0,Y 203.871,Z 250.31,A -85,B 0,C 180,E1 -22021.076,E2 -22021.076} C_VEL
LIN {X 0,Y 202.973,Z 256.091,A -85,B 0,C 180,E1 -22021.298,E2 -22021.298} C_VEL
LIN {X 0,Y 196.385,Z 274.742,A -85,B 0,C 180,E1 -22021.753,E2 -22021.753} C_VEL
LIN {X 0,Y 195.443,Z 280.522,A -85,B 0,C 180,E1 -22021.986,E2 -22021.986} C_VEL
LIN {X 0,Y 194.327,Z 298.659,A -85,B 0,C 180,E1 -22022.98,E2 -22022.98} C_VEL
LIN {X 0,Y 193.074,Z 311.648,A -85,B 0,C 180,E1 -22024.102,E2 -22024.102} C_VEL
LIN {X 0,Y 191.532,Z 324.352,A -85,B 0,C 180,E1 -22025.621,E2 -22025.621} C_VEL
LIN {X 0,Y 189.838,Z 336.408,A -85,B 0,C 180,E1 -22027.527,E2 -22027.527} C_VEL
LIN {X 0,Y 188.092,Z 347.771,A -85,B 0,C 180,E1 -22029.831,E2 -22029.831} C_VEL
LIN {X 0,Y 186.537,Z 358.068,A -85,B 0,C 180,E1 -22032.46,E2 -22032.46} C_VEL
LIN {X 0,Y 185.255,Z 366.556,A -85,B 0,C 180,E1 -22035.165,E2 -22035.165} C_VEL
LIN {X 0,Y 184.217,Z 374.869,A -85,B 0,C 180,E1 -22038.448,E2 -22038.448} C_VEL
LIN {X 0,Y 183.69,Z 380.493,A -85,B 0,C 180,E1 -22041.199,E2 -22041.199} C_VEL
LIN {X 0,Y 183.41,Z 385.946,A -85,B 0,C 180,E1 -22044.506,E2 -22044.506} C_VEL
LIN {X 0,Y 183.406,Z 390.127,A -85,B 0,C 180,E1 -22047.806,E2 -22047.806} C_VEL
LIN {X 0,Y 183.412,Z 392.283,A -85,B 0,C 180,E1 -22050.002,E2 -22050.002} C_VEL
LIN {X 0,Y 183.334,Z 393.925,A -85,B 0,C 180,E1 -22052.199,E2 -22052.199} C_VEL
LIN {X 0,Y 183.227,Z 395.956,A -85,B 0,C 180,E1 -22056.61,E2 -22056.61} C_VEL
LIN {X 0,Y 183.569,Z 396.39,A -85,B 0,C 180,E1 -22058.811,E2 -22058.811} C_VEL
LIN {X 0,Y 184.945,Z 396.05,A -85,B 0,C 180,E1 -22063.181,E2 -22063.181} C_VEL
LIN {X 0,Y 187.3,Z 394.206,A -85,B 0,C 180,E1 -22067.47,E2 -22067.47} C_VEL
LIN {X 0,Y 188.996,Z 392.717,A -85,B 0,C 180,E1 -22069.555,E2 -22069.555} C_VEL
LIN {X 0,Y 193.249,Z 388.445,A -85,B 0,C 180,E1 -22073.583,E2 -22073.583} C_VEL
LIN {X 0,Y 196.89,Z 384.107,A -85,B 0,C 180,E1 -22076.501,E2 -22076.501} C_VEL
LIN {X 0,Y 201.088,Z 378.693,A -85,B 0,C 180,E1 -22079.296,E2 -22079.296} C_VEL
LIN {X 0,Y 205.984,Z 372.031,A -85,B 0,C 180,E1 -22081.929,E2 -22081.929} C_VEL
LIN {X 0,Y 211.413,Z 363.86,A -85,B 0,C 180,E1 -22084.413,E2 -22084.413} C_VEL
LIN {X 0,Y 216.292,Z 355.604,A -85,B 0,C 180,E1 -22086.372,E2 -22086.372} C_VEL
LIN {X 0,Y 221.959,Z 344.661,A -85,B 0,C 180,E1 -22088.42,E2 -22088.42} C_VEL
LIN {X 0,Y 226.852,Z 333.68,A -85,B 0,C 180,E1 -22090.006,E2 -22090.006} C_VEL
LIN {X 0,Y 231.524,Z 321.311,A -85,B 0,C 180,E1 -22091.319,E2 -22091.319} C_VEL
LIN {X 0,Y 235.554,Z 308.225,A -85,B 0,C 180,E1 -22092.314,E2 -22092.314} C_VEL
LIN {X 0,Y 238.315,Z 295.981,A -85,B 0,C 180,E1 -22093.027,E2 -22093.027} C_VEL
LIN {X 0,Y 241.264,Z 276.117,A -85,B 0,C 180,E1 -22093.859,E2 -22093.859} C_VEL
LIN {X 0,Y 243.396,Z 260.159,A -85,B 0,C 180,E1 -22094.476,E2 -22094.476} C_VEL
LIN {X 0,Y 241.276,Z 253.754,A -85,B 0,C 180,E1 -22096.438,E2 -22096.438} C_VEL
LIN {X 0,Y 239.397,Z 248.851,A -85,B 0,C 180,E1 -22098.458,E2 -22098.458} C_VEL
LIN {X 0,Y 238.014,Z 245.498,A -85,B 0,C 180,E1 -22100.152,E2 -22100.152} C_VEL
LIN {X 0,Y 236.336,Z 241.564,A -85,B 0,C 180,E1 -22102.777,E2 -22102.777} C_VEL
LIN {X 0,Y 235.024,Z 238.6,A -85,B 0,C 180,E1 -22106.163,E2 -22106.163} C_VEL
LIN {X 0,Y 234.743,Z 237.602,A -85,B 0,C 180,E1 -22108.358,E2 -22108.358} C_VEL
LIN {X 0,Y 234.948,Z 237.654,A -85,B 0,C 180,E1 -22111.406,E2 -22111.406} C_VEL
LIN {X 0,Y 236.352,Z 239.597,A -85,B 0,C 180,E1 -22115.254,E2 -22115.254} C_VEL
LIN {X 0,Y 236.953,Z 240.485,A -85,B 0,C 180,E1 -22116.274,E2 -22116.274} C_VEL
LIN {X 0,Y 238.973,Z 244.165,A -85,B 0,C 180,E1 -22119.056,E2 -22119.056} C_VEL
LIN {X 0,Y 241.218,Z 248.62,A -85,B 0,C 180,E1 -22121.397,E2 -22121.397} C_VEL
LIN {X 0,Y 243.272,Z 253.042,A -85,B 0,C 180,E1 -22123.209,E2 -22123.209} C_VEL
LIN {X 0,Y 243.969,Z 254.85,A -85,B 0,C 180,E1 -22123.803,E2 -22123.803} C_VEL
LIN {X 0,Y 239.234,Z 288.353,A -85,B 0,C 180,E1 -22125.11,E2 -22125.11} C_VEL
LIN {X 0,Y 236.438,Z 301.498,A -85,B 0,C 180,E1 -22125.882,E2 -22125.882} C_VEL
LIN {X 0,Y 233.077,Z 313.498,A -85,B 0,C 180,E1 -22126.855,E2 -22126.855} C_VEL
LIN {X 0,Y 228.781,Z 325.725,A -85,B 0,C 180,E1 -22128.19,E2 -22128.19} C_VEL
LIN {X 0,Y 223.973,Z 337.087,A -85,B 0,C 180,E1 -22129.834,E2 -22129.834} C_VEL
LIN {X 0,Y 219.116,Z 346.698,A -85,B 0,C 180,E1 -22131.609,E2 -22131.609} C_VEL
LIN {X 0,Y 213.601,Z 356.272,A -85,B 0,C 180,E1 -22133.862,E2 -22133.862} C_VEL
LIN {X 0,Y 208.707,Z 363.792,A -85,B 0,C 180,E1 -22136.139,E2 -22136.139} C_VEL
LIN {X 0,Y 203.874,Z 370.296,A -85,B 0,C 180,E1 -22138.643,E2 -22138.643} C_VEL
LIN {X 0,Y 198.539,Z 376.766,A -85,B 0,C 180,E1 -22142.029,E2 -22142.029} C_VEL
LIN {X 0,Y 194.4,Z 381.18,A -85,B 0,C 180,E1 -22145.186,E2 -22145.186} C_VEL
LIN {X 0,Y 190.877,Z 384.382,A -85,B 0,C 180,E1 -22148.47,E2 -22148.47} C_VEL
LIN {X 0,Y 188.879,Z 385.906,A -85,B 0,C 180,E1 -22150.723,E2 -22150.723} C_VEL
LIN {X 0,Y 187.247,Z 386.913,A -85,B 0,C 180,E1 -22153.015,E2 -22153.015} C_VEL
LIN {X 0,Y 185.862,Z 387.493,A -85,B 0,C 180,E1 -22155.349,E2 -22155.349} C_VEL
LIN {X 0,Y 184.668,Z 387.585,A -85,B 0,C 180,E1 -22157.924,E2 -22157.924} C_VEL
LIN {X 0,Y 183.871,Z 387.216,A -85,B 0,C 180,E1 -22160.122,E2 -22160.122} C_VEL
LIN {X 0,Y 183.157,Z 386.203,A -85,B 0,C 180,E1 -22162.936,E2 -22162.936} C_VEL
LIN {X 0,Y 182.818,Z 385.001,A -85,B 0,C 180,E1 -22165.017,E2 -22165.017} C_VEL
LIN {X 0,Y 182.72,Z 381.877,A -85,B 0,C 180,E1 -22168.788,E2 -22168.788} C_VEL
LIN {X 0,Y 183.04,Z 377.458,A -85,B 0,C 180,E1 -22172.517,E2 -22172.517} C_VEL
LIN {X 0,Y 183.552,Z 372.31,A -85,B 0,C 180,E1 -22175.807,E2 -22175.807} C_VEL
LIN {X 0,Y 184.279,Z 366.019,A -85,B 0,C 180,E1 -22178.998,E2 -22178.998} C_VEL
LIN {X 0,Y 185.395,Z 357.864,A -85,B 0,C 180,E1 -22182.289,E2 -22182.289} C_VEL
LIN {X 0,Y 186.74,Z 348.881,A -85,B 0,C 180,E1 -22185.198,E2 -22185.198} C_VEL
LIN {X 0,Y 188.202,Z 339.121,A -85,B 0,C 180,E1 -22187.763,E2 -22187.763} C_VEL
LIN {X 0,Y 189.964,Z 327.691,A -85,B 0,C 180,E1 -22190.147,E2 -22190.147} C_VEL
LIN {X 0,Y 191.719,Z 315.024,A -85,B 0,C 180,E1 -22192.209,E2 -22192.209} C_VEL
LIN {X 0,Y 193.245,Z 301.688,A -85,B 0,C 180,E1 -22193.829,E2 -22193.829} C_VEL
LIN {X 0,Y 194.368,Z 288.193,A -85,B 0,C 180,E1 -22195.018,E2 -22195.018} C_VEL
LIN {X 0,Y 195.468,Z 270.942,A -85,B 0,C 180,E1 -22195.961,E2 -22195.961} C_VEL
LIN {X 0,Y 198.341,Z 217.975,A -85,B 0,C 180,E1 -22198.488,E2 -22198.488} C_VEL
LIN {X 0,Y 191.152,Z 195.18,A -85,B 0,C 180,E1 -22200.408,E2 -22200.408} C_VEL
LIN {X 0,Y 185.572,Z 180.439,A -85,B 0,C 180,E1 -22201.82,E2 -22201.82} C_VEL
LIN {X 0,Y 185.549,Z 180.372,A -85,B 0,C 180,E1 -22205.375,E2 -22205.375} C_VEL
LIN {X 0,Y 185.63,Z 180.362,A -85,B 0,C 180,E1 -22211.177,E2 -22211.177} C_VEL
LIN {X 0,Y 185.704,Z 180.353,A -85,B 0,C 180,E1 -22216.873,E2 -22216.873} C_VEL
LIN {X 0,Y 185.979,Z 180.317,A -85,B 0,C 180,E1 -22221.304,E2 -22221.304} C_VEL
LIN {X 0,Y 186.18,Z 180.293,A -85,B 0,C 180,E1 -22227.835,E2 -22227.835} C_VEL
LIN {X 0,Y 186.383,Z 180.265,A -85,B 0,C 180,E1 -22229.998,E2 -22229.998} C_VEL
LIN {X 0,Y 185.887,Z 180.329,A -85,B 0,C 180,E1 -22234.335,E2 -22234.335} C_VEL
LIN {X 0,Y 185.974,Z 180.313,A -85,B 0,C 180,E1 -22238.692,E2 -22238.692} C_VEL
LIN {X 0,Y 185.701,Z 180.353,A -85,B 0,C 180,E1 -22243.123,E2 -22243.123} C_VEL
LIN {X 0,Y 185.626,Z 180.36,A -85,B 0,C 180,E1 -22248.819,E2 -22248.819} C_VEL
LIN {X 0,Y 185.544,Z 180.369,A -85,B 0,C 180,E1 -22254.621,E2 -22254.621} C_VEL
LIN {X 0,Y 185.543,Z 180.373,A -85,B 0,C 180,E1 -22259.497,E2 -22259.497} C_VEL
LIN {X 0,Y 185.495,Z 180.375,A -85,B 0,C 180,E1 -22264.63,E2 -22264.63} C_VEL
LIN {X 0,Y 185.497,Z 180.379,A -85,B 0,C 180,E1 -22267.312,E2 -22267.312} C_VEL
LIN {X 0,Y 185.459,Z 180.382,A -85,B 0,C 180,E1 -22270.719,E2 -22270.719} C_VEL
LIN {X 0,Y 185.452,Z 180.383,A -85,B 0,C 180,E1 -22276.054,E2 -22276.054} C_VEL
LIN {X 0,Y 185.452,Z 180.379,A -85,B 0,C 180,E1 -22279.89,E2 -22279.89} C_VEL
LIN {X 0,Y 185.496,Z 180.379,A -85,B 0,C 180,E1 -22282.712,E2 -22282.712} C_VEL
LIN {X 0,Y 185.526,Z 180.371,A -85,B 0,C 180,E1 -22287.971,E2 -22287.971} C_VEL
LIN {X 0,Y 185.542,Z 180.372,A -85,B 0,C 180,E1 -22290.594,E2 -22290.594} C_VEL
LIN {X 0,Y 185.557,Z 180.368,A -85,B 0,C 180,E1 -22295.378,E2 -22295.378} C_VEL
LIN {X 0,Y 185.619,Z 180.362,A -85,B 0,C 180,E1 -22301.178,E2 -22301.178} C_VEL
LIN {X 0,Y 185.693,Z 180.352,A -85,B 0,C 180,E1 -22306.874,E2 -22306.874} C_VEL
LIN {X 0,Y 185.969,Z 180.318,A -85,B 0,C 180,E1 -22311.305,E2 -22311.305} C_VEL
LIN {X 0,Y 186.169,Z 180.296,A -85,B 0,C 180,E1 -22317.836,E2 -22317.836} C_VEL
LIN {X 0,Y 186.373,Z 180.269,A -85,B 0,C 180,E1 -22320,E2 -22320} C_VEL
LIN {X 0,Y 185.877,Z 180.33,A -85,B 0,C 180,E1 -22324.336,E2 -22324.336} C_VEL
LIN {X 0,Y 185.965,Z 180.317,A -85,B 0,C 180,E1 -22328.694,E2 -22328.694} C_VEL
LIN {X 0,Y 185.692,Z 180.352,A -85,B 0,C 180,E1 -22333.125,E2 -22333.125} C_VEL
LIN {X 0,Y 185.618,Z 180.358,A -85,B 0,C 180,E1 -22338.821,E2 -22338.821} C_VEL
LIN {X 0,Y 185.538,Z 180.372,A -85,B 0,C 180,E1 -22344.624,E2 -22344.624} C_VEL
LIN {X 0,Y 185.537,Z 180.374,A -85,B 0,C 180,E1 -22349.5,E2 -22349.5} C_VEL
LIN {X 0,Y 185.491,Z 180.377,A -85,B 0,C 180,E1 -22354.634,E2 -22354.634} C_VEL
LIN {X 0,Y 185.494,Z 180.376,A -85,B 0,C 180,E1 -22357.316,E2 -22357.316} C_VEL
LIN {X 0,Y 185.455,Z 180.384,A -85,B 0,C 180,E1 -22360.722,E2 -22360.722} C_VEL
LIN {X 0,Y 185.45,Z 180.385,A -85,B 0,C 180,E1 -22366.058,E2 -22366.058} C_VEL
